# B&R Automation Studio project GAT (part 7)

#### Variables.var
```iecst
VAR
	MC_BR_ProcessConfig_AX : MC_BR_ProcessConfig; (*Function block to read and write the axis configuration*)
	MC_BR_ProcessConfig_ACP : MC_BR_ProcessConfig; (*Function block to read and write the ACOPOS configuration*)
	BaseAxConfig : ARRAY[0..1] OF McCfgAxType; (*Acopos configuration*)
	AcpAxConfig : ARRAY[0..1] OF McCfgAcpAxType; (*Acopos configuration*)
	uSelectedAxis : USINT; (*Selected Axis index*)
	sAxFeatures1 : ARRAY[0..2] OF STRING[255]; (*Axis features*)
	sAxFeatures2 : ARRAY[0..2] OF STRING[255]; (*Axis features*)
	uState : UINT; (*Read/Write state machine status*)
	bReadConfig : BOOL; (*Read config command*)
	bWriteConfig : BOOL; (*Write Acopos config command*)
	bSuccessRead : BOOL; (*Read config succeeded*)
	bErrorRead : BOOL; (*Read config failed*)
	bErrorWrite : BOOL; (*Write config failed*)
	bSuccessWrite : BOOL; (*Write config succeeded*)
	bSysReboot : BOOL;
	MpRecipeRegPar_M : ARRAY[0..3] OF MpRecipeRegPar;
	MC_BR_ProcessParam_ACP : MC_BR_ProcessParam;
END_VAR
```

#### Main.st
```iecst
//*********************************************************************************
//* Copyright: B&R Industrial Automation GmbH
//* This task let's the OEM change the ACOPOS configuration via the HMI
//*********************************************************************************

PROGRAM _INIT
	// FUB configuration: MC_BR_ProcessConfig for persistent configuration changes, MC_BR_ProcessParam for online configuration changes
    MC_BR_ProcessConfig_ACP.DataType := mcCFG_ACP_AX;

	AcpAxConfig[0].AxisFeatures.FeatureReference.DataAddress := ADR(AxFeatures1);
	AcpAxConfig[0].AxisFeatures.FeatureReference.NumberOfArrayElements := 3;
	AcpAxConfig[1].AxisFeatures.FeatureReference.DataAddress := ADR(AxFeatures2);
	AcpAxConfig[1].AxisFeatures.FeatureReference.NumberOfArrayElements := 3;

	MC_BR_ProcessConfig_AX.DataType := mcCFG_AX;

	MC_BR_ProcessParam_ACP.ExecutionMode := mcEM_IMMEDIATELY;
	MC_BR_ProcessParam_ACP.Mode := mcPPM_WRITE;

	// Register "Machine" category PVs
	MpRecipeRegPar_M[0].MpLink := ADR(gMpLinkRecipeXml);
	MpRecipeRegPar_M[0].Enable := TRUE;
	MpRecipeRegPar_M[0].Category := ADR('Machine');
	MpRecipeRegPar_M[0].PVName := ADR('ProcessCon:AcpAxConfig');
	MpRecipeRegPar_M[1].MpLink := ADR(gMpLinkRecipeXml);
	MpRecipeRegPar_M[1].Enable := TRUE;
	MpRecipeRegPar_M[1].Category := ADR('Machine');
	MpRecipeRegPar_M[1].PVName := ADR('ProcessCon:BaseAxConfig');
	MpRecipeRegPar_M[2].MpLink := ADR(gMpLinkRecipeXml);
	MpRecipeRegPar_M[2].Enable := TRUE;
	MpRecipeRegPar_M[2].Category := ADR('Machine');
	MpRecipeRegPar_M[2].PVName := ADR('ProcessCon:sAxFeatures1');
	MpRecipeRegPar_M[3].MpLink := ADR(gMpLinkRecipeXml);
	MpRecipeRegPar_M[3].Enable := TRUE;
	MpRecipeRegPar_M[3].Category := ADR('Machine');
	MpRecipeRegPar_M[3].PVName := ADR('ProcessCon:sAxFeatures2');

	// Activate RegPar FUBs
	WHILE NOT MpRecipeRegPar_M[0].Active DO
		MpRecipeRegPar_M[0]();
	END_WHILE
	WHILE NOT MpRecipeRegPar_M[1].Active DO
		MpRecipeRegPar_M[1]();
	END_WHILE
	WHILE NOT MpRecipeRegPar_M[2].Active DO
		MpRecipeRegPar_M[2]();
	END_WHILE
	WHILE NOT MpRecipeRegPar_M[3].Active DO
		MpRecipeRegPar_M[3]();
	END_WHILE

	// Trigger first read
	ReadConfig := TRUE;
	State := 0;
END_PROGRAM

PROGRAM _CYCLIC
	// Read/Write state machine
	CASE State OF
        0:
            // Idle
			IF MpRecipeRegPar_M[0].UpdateNotification THEN
				// Reset the address of sAxFeatures1/2
				AcpAxConfig[0].AxisFeatures.FeatureReference.DataAddress := ADR(AxFeatures1);
				AcpAxConfig[0].AxisFeatures.FeatureReference.NumberOfArrayElements := 3;
				AcpAxConfig[1].AxisFeatures.FeatureReference.DataAddress := ADR(AxFeatures2);
				AcpAxConfig[1].AxisFeatures.FeatureReference.NumberOfArrayElements := 3;

				// Write the configuration
				SelectedAxis := 0;
				WriteConfig := TRUE;
				ReadConfig := FALSE;
			ELSIF ReadConfig THEN
				// Set axis dependend configuration name
				IF SelectedAxis = 0 THEN
					brsstrcpy(ADR(MC_BR_ProcessConfig_ACP.Name), ADR('IF1.ST1/DriveConfiguration/Channel1'));
				ELSE
					brsstrcpy(ADR(MC_BR_ProcessConfig_ACP.Name), ADR('IF1.ST1/DriveConfiguration/Channel2'));
				END_IF
				AcpAxConfig[0].AxisFeatures.FeatureReference.DataAddress := ADR(AxFeatures1);
				AcpAxConfig[0].AxisFeatures.FeatureReference.NumberOfArrayElements := 3;
				AcpAxConfig[1].AxisFeatures.FeatureReference.DataAddress := ADR(AxFeatures2);
				AcpAxConfig[1].AxisFeatures.FeatureReference.NumberOfArrayElements := 3;

				MC_BR_ProcessConfig_ACP.DataAddress := ADR(AcpAxConfig[SelectedAxis]);
				MC_BR_ProcessConfig_AX.DataAddress := ADR(BaseAxConfig[SelectedAxis]);
				// Start loading
				MC_BR_ProcessConfig_ACP.Mode := mcPCM_LOAD;
				MC_BR_ProcessConfig_ACP.Execute := TRUE;
				ErrorRead := FALSE;
				SuccessRead := FALSE;
				State := 10;
			ELSIF WriteConfig THEN
				// Set axis dependend configuration name
				IF SelectedAxis = 0 THEN
					brsstrcpy(ADR(MC_BR_ProcessConfig_ACP.Name), ADR('IF1.ST1/DriveConfiguration/Channel1'));
					MC_BR_ProcessParam_ACP.Component := ADR(gAxisMaster);
				ELSE
					brsstrcpy(ADR(MC_BR_ProcessConfig_ACP.Name), ADR('IF1.ST1/DriveConfiguration/Channel2'));
					MC_BR_ProcessParam_ACP.Component := ADR(gAxisSlave);
				END_IF
				MC_BR_ProcessConfig_ACP.DataAddress := ADR(AcpAxConfig[SelectedAxis]);
				MC_BR_ProcessConfig_AX.DataAddress := ADR(BaseAxConfig[SelectedAxis]);
                MC_BR_ProcessParam_ACP.DataAddress := ADR(AcpAxConfig[SelectedAxis].MechanicalElements);
                // mcCFG_ACP_AX is not supported yet, therefore, transfer mech elements and homing parameters in two steps
				MC_BR_ProcessParam_ACP.DataType := mcCFG_ACP_MECH_ELM;
				// Copy direct homing position into the used homing mode, HMI is bound to direct homing position
				CASE AcpAxConfig[SelectedAxis].Homing.Mode.Type OF
					mcAHM_ABS:
						AcpAxConfig[SelectedAxis].Homing.Mode.Absolute.Position := AcpAxConfig[SelectedAxis].Homing.Mode.Direct.Position;
					mcAHM_ABS_CORR:
						AcpAxConfig[SelectedAxis].Homing.Mode.AbsoluteCorrection.Position := AcpAxConfig[SelectedAxis].Homing.Mode.Direct.Position;
					mcAHM_ABS_SW:
						AcpAxConfig[SelectedAxis].Homing.Mode.AbsoluteSwitch.Position := AcpAxConfig[SelectedAxis].Homing.Mode.Direct.Position;
					mcAHM_BLK_LAG_ERR:
						AcpAxConfig[SelectedAxis].Homing.Mode.BlockLagError.Position := AcpAxConfig[SelectedAxis].Homing.Mode.Direct.Position;
                    mcAHM_BLK_TORQ:
                        AcpAxConfig[SelectedAxis].Homing.Mode.BlockTorque.Position := AcpAxConfig[SelectedAxis].Homing.Mode.Direct.Position;
					mcAHM_DIST_C_MARKS:
						AcpAxConfig[SelectedAxis].Homing.Mode.DistanceCodedMarks.Position := AcpAxConfig[SelectedAxis].Homing.Mode.Direct.Position;
					mcAHM_DIST_C_MARKS_CORR:
						AcpAxConfig[SelectedAxis].Homing.Mode.DistanceCodedMarksCorrection.Position := AcpAxConfig[SelectedAxis].Homing.Mode.Direct.Position;
					mcAHM_LIM_SW:
						AcpAxConfig[SelectedAxis].Homing.Mode.LimitSwitch.Position := AcpAxConfig[SelectedAxis].Homing.Mode.Direct.Position;
					mcAHM_SW_GATE:
						AcpAxConfig[SelectedAxis].Homing.Mode.SwitchGate.Position := AcpAxConfig[SelectedAxis].Homing.Mode.Direct.Position;
				END_CASE;
				MC_BR_ProcessConfig_ACP.Mode := mcPCM_SAVE;
				MC_BR_ProcessConfig_ACP.Execute := TRUE;
				MC_BR_ProcessConfig_AX.Mode := mcPCM_SAVE;
				MC_BR_ProcessConfig_AX.Execute := TRUE;
				MC_BR_ProcessParam_ACP.Execute := TRUE;
				ErrorWrite := FALSE;
				SuccessWrite := FALSE;
				State := 20;
			END_IF

        10:
            // Read config
			IF MC_BR_ProcessConfig_ACP.Done OR MC_BR_ProcessConfig_ACP.Error THEN
				MC_BR_ProcessConfig_ACP.Execute := FALSE;
				// Copy homing position into the direct homing position, HMI is bound to direct homing position
				CASE AcpAxConfig[SelectedAxis].Homing.Mode.Type OF
					mcAHM_ABS:
						AcpAxConfig[SelectedAxis].Homing.Mode.Direct.Position := AcpAxConfig[SelectedAxis].Homing.Mode.Absolute.Position;
					mcAHM_ABS_CORR:
						AcpAxConfig[SelectedAxis].Homing.Mode.Direct.Position := AcpAxConfig[SelectedAxis].Homing.Mode.AbsoluteCorrection.Position;
					mcAHM_ABS_SW:
						AcpAxConfig[SelectedAxis].Homing.Mode.Direct.Position := AcpAxConfig[SelectedAxis].Homing.Mode.AbsoluteSwitch.Position;
					mcAHM_BLK_LAG_ERR:
						AcpAxConfig[SelectedAxis].Homing.Mode.Direct.Position := AcpAxConfig[SelectedAxis].Homing.Mode.BlockLagError.Position;
					mcAHM_BLK_TORQ:
						AcpAxConfig[SelectedAxis].Homing.Mode.Direct.Position := AcpAxConfig[SelectedAxis].Homing.Mode.BlockTorque.Position;
					mcAHM_DIST_C_MARKS:
						AcpAxConfig[SelectedAxis].Homing.Mode.Direct.Position := AcpAxConfig[SelectedAxis].Homing.Mode.DistanceCodedMarks.Position;
					mcAHM_DIST_C_MARKS_CORR:
						AcpAxConfig[SelectedAxis].Homing.Mode.Direct.Position := AcpAxConfig[SelectedAxis].Homing.Mode.DistanceCodedMarksCorrection.Position;
					mcAHM_LIM_SW:
						AcpAxConfig[SelectedAxis].Homing.Mode.Direct.Position := AcpAxConfig[SelectedAxis].Homing.Mode.LimitSwitch.Position;
					mcAHM_SW_GATE:
						AcpAxConfig[SelectedAxis].Homing.Mode.Direct.Position := AcpAxConfig[SelectedAxis].Homing.Mode.SwitchGate.Position;
				END_CASE;
				brsstrcpy(ADR(MC_BR_ProcessConfig_AX.Name), ADR(AcpAxConfig[SelectedAxis].AxisReference.Name));
				MC_BR_ProcessConfig_AX.Mode := mcPCM_LOAD;
				MC_BR_ProcessConfig_AX.Execute := TRUE;
				ErrorRead := FALSE;
				SuccessRead := TRUE;
				State := 11;
			ELSIF MC_BR_ProcessConfig_ACP.Error THEN
				MC_BR_ProcessConfig_ACP.Execute := FALSE;
				ErrorRead := TRUE;
				SuccessRead := FALSE;
				ReadConfig := FALSE;
				State := 0;
			END_IF

        11:
            // Read axis config
			IF MC_BR_ProcessConfig_AX.Done OR MC_BR_ProcessConfig_AX.Error THEN
				MC_BR_ProcessConfig_AX.Execute := FALSE;
				ErrorRead := MC_BR_ProcessConfig_AX.Error;
				SuccessRead := NOT bErrorRead;
				IF SelectedAxis = 0 THEN
					SelectedAxis := 1;
				ELSE
					ReadConfig := FALSE;
				END_IF
				State := 0;
			END_IF

        20:
            // Write config
			IF (MC_BR_ProcessConfig_ACP.Done OR MC_BR_ProcessConfig_ACP.Error)
				AND (MC_BR_ProcessConfig_AX.Done OR MC_BR_ProcessConfig_AX.Error)
				AND (MC_BR_ProcessParam_ACP.Done OR MC_BR_ProcessParam_ACP.Error) THEN
				MC_BR_ProcessConfig_ACP.Execute := FALSE;
				MC_BR_ProcessConfig_AX.Execute := FALSE;
				MC_BR_ProcessParam_ACP.Execute := FALSE;
				ErrorWrite := MC_BR_ProcessConfig_ACP.Error OR MC_BR_ProcessConfig_AX.Error OR MC_BR_ProcessParam_ACP.Error;
				SuccessWrite := NOT ErrorWrite;
				State := 21;
			END_IF

        21:
            // Write Homing config
			MC_BR_ProcessParam_ACP.DataAddress := ADR(AcpAxConfig[SelectedAxis].Homing);// mcCFG_ACP_AX is not supported yet, therefore, transfer mech elements and homing parameters in two steps
			MC_BR_ProcessParam_ACP.DataType := mcCFG_ACP_HOME;
			MC_BR_ProcessParam_ACP.Execute := TRUE;
			IF MC_BR_ProcessParam_ACP.Done OR MC_BR_ProcessParam_ACP.Error THEN
				MC_BR_ProcessParam_ACP.Execute := FALSE;
				ErrorWrite := bErrorWrite OR MC_BR_ProcessParam_ACP.Error;
				SuccessWrite := NOT bErrorWrite;
				State := 0;
				// Update the second axis, or finish
				IF SelectedAxis = 0 THEN
					SelectedAxis := 1;
				ELSE
					WriteConfig := FALSE;
				END_IF
			END_IF
	END_CASE;

	// PLC reboot
	IF SysReboot THEN
		SYSreset(TRUE, 1);
	END_IF

	// Function block calls
	MC_BR_ProcessConfig_ACP();
	MC_BR_ProcessConfig_AX();
	MC_BR_ProcessParam_ACP();
	MpRecipeRegPar_M[0]();
	MpRecipeRegPar_M[1]();
	MpRecipeRegPar_M[2]();
	MpRecipeRegPar_M[3]();
END_PROGRAM

PROGRAM _EXIT
	// Release mplink
	MpRecipeRegPar_M[0].Enable := FALSE;
	MpRecipeRegPar_M[1].Enable := FALSE;
	MpRecipeRegPar_M[2].Enable := FALSE;
	MpRecipeRegPar_M[3].Enable := FALSE;
	MpRecipeRegPar_M[0]();
	MpRecipeRegPar_M[1]();
	MpRecipeRegPar_M[2]();
	MpRecipeRegPar_M[3]();
END_PROGRAM
```

### Program Logical/Infrastructure/SysServices/IoBrowser (IEC) - Task to read the IO module structure and display the IO channels

#### Variables.var
```iecst
(*Io process related variables*)
VAR
	GatIoForcingHandler_0 : GatIoForcingHandler; (*Function block for Io handling (browser & forcing)*)
	IoModules : ARRAY[0..gatMAX_IDX_IO_MODULES] OF GatIoModulesType;
	pIoChannelTemp : REFERENCE TO GatIoChannelType;
	pIoChannel : REFERENCE TO GatIoChannelType;
END_VAR
(*Helper variables for mappView*)
VAR
	sStationList : ARRAY[0..gatMAX_IDX_IO_MODULES] OF STRING[80];
	sModuleList : ARRAY[0..gatMAX_IDX_IO_MODULES] OF STRING[80];
	sIoChannelList : ARRAY[0..gatMAX_IDX_IO_CHANNELS] OF STRING[80];
	sIoPvList : ARRAY[0..gatMAX_IDX_IO_CHANNELS] OF STRING[80];
	sIoValueList : ARRAY[0..gatMAX_IDX_IO_CHANNELS] OF STRING[20];
	iIoValueList : ARRAY[0..gatMAX_IDX_IO_CHANNELS] OF DINT;
	uStationIdx : UINT;
	uModuleIdx : UINT;
	uChannelIdx : UINT;
	sSelectedStation : STRING[80];
	uSelectedStation : UINT;
	uLastSelectedStation : UINT;
	uSelectedModule : UINT;
	uLastSelectedModule : UINT;
	uSelectedChannel : UINT;
	uLastSelectedChannel : UINT;
	sTableConfigChannels : STRING[200];
	sTableConfigStations : STRING[200];
	sTableConfig : STRING[200];
	sTempStationPath : STRING[80];
	bLastModuleInvisible : BOOL;
END_VAR
```

#### Main.st
```iecst
//*********************************************************************************
//* Copyright: B&R Industrial Automation GmbH
//* This program provides an Io browser and the related interface for
//* mappView widgets.
//*********************************************************************************

PROGRAM _INIT
	// Init Io handler
	GatIoForcingHandler_0.Enable := TRUE;
	GatIoForcingHandler_0.SelectedRefreshMode := TRUE;
	GatIoForcingHandler_0.IoModules := ADR(IoModules);

	// Init refresh selection
	FOR ChannelIdx := 0 TO gatMAX_IDX_IO_CHANNELS DO
		IoModules[0].IoChannels[ChannelIdx].IoForcing.RefreshActualValue := TRUE;
	END_FOR

	// Init Table configs for mappView
	brsstrcpy(ADR(TableConfig), ADR('{ "specRows": [{"from":0,"to":19, "visible":false}]}'));
	brsstrcpy(ADR(TableConfigStations), ADR('{ "specRows": [{"from":0,"to":19, "visible":false}]}'));
	brsstrcpy(ADR(TableConfigChannels), ADR('{ "specRows": [{"from":0,"to":31, "visible":false}]}'));

	// Init pointers
	IoChannel ACCESS ADR(IoModules[0].IoChannels[0]);
	IoChannelTemp ACCESS ADR(IoModules[0].IoChannels[0]);
END_PROGRAM

PROGRAM _CYCLIC
	// Action to prepare all necessary table configs etc for mappView according to the station/module selection
	mappViewAction;

	// Function block call
	GatIoForcingHandler_0();
END_PROGRAM

PROGRAM _EXIT
	// Disabled function block call
	GatIoForcingHandler_0.Enable := FALSE;
	GatIoForcingHandler_0();
END_PROGRAM
```

#### mappViewAction.st
```iecst
//*********************************************************************************
//* Copyright: B&R Industrial Automation GmbH
//* This action sets all the strings and pointers so that the mappView page can
//* present the IO information in a user friendly way
//********************************************************************************

ACTION mappViewAction:
	// Set pointers to the correct Forcing handler for easier interface to HMI
	IF (SelectedModule <> LastSelectedModule) OR (SelectedChannel <> LastSelectedChannel) THEN
		// Check range
		IF (SelectedModule <= gatMAX_IDX_IO_MODULES) AND (SelectedChannel <= gatMAX_IDX_IO_MODULES) THEN
			IF SelectedChannel >= IoModules[SelectedModule].NrOfIoChannels THEN
				SelectedChannel := 0;
			END_IF
			IoChannel ACCESS ADR(IoModules[SelectedModule].IoChannels[SelectedChannel]);
			IoChannelTemp ACCESS ADR(IoModules[SelectedModule].IoChannels[SelectedChannel]);
			brsmemset(ADR(IoChannelList), 0, SIZEOF(IoChannelList));
			brsmemset(ADR(IoPvList), 0, SIZEOF(IoPvList));
			brsmemset(ADR(IoValueList), 0, SIZEOF(IoValueList));
			brsmemset(ADR(TableConfigChannels), 0, SIZEOF(TableConfigChannels));
			FOR ChannelIdx := 0 TO gatMAX_IDX_IO_CHANNELS DO
				brsstrcpy(ADR(IoChannelList[ChannelIdx]), ADR(IoModules[SelectedModule].IoChannels[ChannelIdx].ChannelName));
				IF brsstrlen(ADR(IoChannelList[ChannelIdx])) = 0 THEN
					// Configure visible table entries
					brsstrcpy(ADR(TableConfigChannels), ADR('{ "specRows": [{"from":'));
					brsitoa(ChannelIdx, ADR(TableConfigChannels) + brsstrlen(ADR(TableConfigChannels)));
					brsstrcat(ADR(TableConfigChannels),  ADR(',"to":31, "visible":false}]}'));
					EXIT;
				END_IF
				brsstrcpy(ADR(IoPvList[ChannelIdx]), ADR('$$IAT/Audit/DP/'));
				IF brsstrlen(ADR(IoModules[SelectedModule].IoChannels[ChannelIdx].PvName)) = 0 THEN
					brsstrcat(ADR(IoPvList[ChannelIdx]), ADR('None'));
				ELSE
					brsstrcat(ADR(IoPvList[ChannelIdx]), ADR(IoModules[SelectedModule].IoChannels[ChannelIdx].PvName));
				END_IF
			END_FOR
			LastSelectedModule := SelectedModule;
			LastSelectedChannel := SelectedChannel;
		END_IF
		// Set Io refresh flags
		FOR ModuleIdx := 0 TO gatMAX_IDX_IO_MODULES DO
			FOR ChannelIdx := 0 TO gatMAX_IDX_IO_CHANNELS DO
				IoModules[ModuleIdx].IoChannels[ChannelIdx].IoForcing.RefreshActualValue := (ModuleIdx = SelectedModule);
			END_FOR
		END_FOR
	END_IF

	// Update IO values
	FOR ChannelIdx := 0 TO gatMAX_IDX_IO_CHANNELS DO
		IF IoModules[SelectedModule].IoChannels[ChannelIdx].IoForcing.ActualValue > 32767 THEN
			IoValueList[ChannelIdx] := IoModules[SelectedModule].IoChannels[ChannelIdx].IoForcing.ActualValue - 65536;
		ELSE
			IoValueList[ChannelIdx] := IoModules[SelectedModule].IoChannels[ChannelIdx].IoForcing.ActualValue;
		END_IF
		CASE IoModules[SelectedModule].IoChannels[ChannelIdx].Type OF
			IO_DIG_INPUT, IO_DIG_OUTPUT:
				IF (IoModules[SelectedModule].IoChannels[ChannelIdx].IoForcing.ActualValue = 1) THEN
					brsstrcpy(ADR(IoValueListString[ChannelIdx]), ADR('ON'));
				ELSE
					brsstrcpy(ADR(IoValueListString[ChannelIdx]), ADR('OFF'));
				END_IF
			IO_ANA_INPUT, IO_ANA_OUTPUT, IO_PWM_OUTPUT:
				brsftoa(DINT_TO_REAL(REAL_TO_DINT(DINT_TO_REAL(IoValueList[ChannelIdx]) / 32.767)) / 10, ADR(IoValueListString[ChannelIdx]));
				brsstrcat(ADR(IoValueListString[ChannelIdx]), ADR(' %'));
			IO_TEMP_INPUT:
				brsftoa(DINT_TO_REAL(IoValueList[ChannelIdx]) / 10, ADR(IoValueListString[ChannelIdx]));
				brsstrcat(ADR(IoValueListString[ChannelIdx]), ADR(' C'));
			ELSE
				brsitoa(IoValueList[ChannelIdx], ADR(IoValueListString[ChannelIdx]));
		END_CASE
	END_FOR

	// Init Io Module list when handler is ready
	IF EDGEPOS(GatIoForcingHandler_0.Ready) THEN
		brsmemset(ADR(TableConfigStations), 0, SIZEOF(TableConfig));
		brsmemset(ADR(StationList), 0, SIZEOF(StationList));
		// Init station list
		FOR ModuleIdx := 0 TO gatMAX_IDX_IO_MODULES DO
			IF FIND(RIGHT(IoModules[ModuleIdx].ModulePath, 6), '.') > 0 THEN
				brsmemset(ADR(TempStationPath), 0, SIZEOF(TempStationPath));
				brsstrcpy(ADR(TempStationPath), ADR('$$IAT/IoStations/'));
				brsmemcpy(ADR(TempStationPath) + brsstrlen(ADR(TempStationPath)), ADR(IoModules[ModuleIdx].ModulePath), brsstrlen(ADR(IoModules[ModuleIdx].ModulePath)) - 7 + FIND(RIGHT(IoModules[ModuleIdx].ModulePath, 6), '.'));
			END_IF
			FOR StationIdx := 0 TO gatMAX_IDX_IO_MODULES DO
				IF brsstrcmp(ADR(StationList[StationIdx]), ADR(TempStationPath)) = 0 THEN
					// Station already registered
					EXIT;
				END_IF
				IF brsstrlen(ADR(StationList[StationIdx])) = 0 THEN
					// Reached end of list, add new station
					brsstrcpy(ADR(StationList[StationIdx]), ADR(TempStationPath));
					EXIT;
				END_IF
			END_FOR
		END_FOR
		// Set station table configuration
		FOR StationIdx := 0 TO gatMAX_IDX_IO_MODULES DO
			IF brsstrlen(ADR(StationList[StationIdx])) = 0 THEN
				brsstrcpy(ADR(TableConfigStations), ADR('{ "specRows": [{"from":'));
				brsitoa(StationIdx, ADR(TableConfigStations) + brsstrlen(ADR(TableConfigStations)));
				brsstrcat(ADR(TableConfigStations),  ADR(',"to":'));
				brsstrcat(ADR(TableConfigStations),  ADR('19, "visible":false}]}'));
				EXIT;
			END_IF
		END_FOR
		// Trigger station selection
		SelectedStationIndex := 0;
		LastSelectedStationIndex := 1;
	END_IF

	// Init Module list after station selection
	IF SelectedStationIndex <> LastSelectedStationIndex THEN
		brsmemset(ADR(TableConfig), 0, SIZEOF(TableConfig));
		brsmemset(ADR(ModuleList), 0, SIZEOF(ModuleList));
		brsmemset(ADR(SelectedStation), 0, SIZEOF(SelectedStation));
		brsstrcpy(ADR(SelectedStation), ADR(StationList[SelectedStationIndex]) + brsstrlen(ADR('$$IAT/IoStations/')));
		// Init module list
		brsmemset(ADR(TableConfig), 0, SIZEOF(TableConfig));
		LastModuleInvisible := FALSE;
		FOR ModuleIdx := 0 TO gatMAX_IDX_IO_MODULES DO
			brsstrcpy(ADR(ModuleList[ModuleIdx]), ADR(IoModules[ModuleIdx].ModuleName));
			IF (FIND(IoModules[ModuleIdx].ModulePath, SelectedStation) = 0) THEN
				// Wrong station, make station invisible
				IF NOT LastModuleInvisible THEN
					IF brsstrlen(ADR(TableConfig)) = 0 THEN
						brsstrcpy(ADR(TableConfig), ADR('{ "specRows": [{"from":'));
					ELSE
						brsstrcat(ADR(TableConfig), ADR(', {"from":'));
					END_IF
					brsitoa(ModuleIdx, ADR(TableConfig) + brsstrlen(ADR(TableConfig)));
					brsstrcat(ADR(TableConfig),  ADR(',"to":'));
				END_IF
				LastModuleInvisible := TRUE;
			ELSE
				// Correct station, make module visible and select it if it's the first module of the station
				IF SelectedModule = LastSelectedModule THEN
					SelectedModule := ModuleIdx;
					LastSelectedModule := SelectedModule + 1;
				END_IF
				IF LastModuleInvisible THEN
					brsitoa(ModuleIdx - 1, ADR(TableConfig) + brsstrlen(ADR(TableConfig)));
					brsstrcat(ADR(TableConfig),  ADR(', "visible":false}'));
				END_IF
				LastModuleInvisible := FALSE;
			END_IF
			IF brsstrlen(ADR(ModuleList[ModuleIdx])) = 0 THEN
				// Reached end of modules, make rest of list invisible
				IF NOT LastModuleInvisible THEN
					IF brsstrlen(ADR(TableConfig)) = 0 THEN
						brsstrcpy(ADR(TableConfig), ADR('{ "specRows": [{"from":'));
					ELSE
						brsstrcat(ADR(TableConfig), ADR(', {"from":'));
					END_IF
					brsitoa(ModuleIdx, ADR(TableConfig) + brsstrlen(ADR(TableConfig)));
					brsstrcat(ADR(TableConfig),  ADR(',"to":'));
				END_IF
				brsstrcat(ADR(TableConfig),  ADR('19, "visible":false}]}'));
				EXIT;
			ELSIF ModuleIdx = gatMAX_IDX_IO_MODULES THEN
				// Reached end of modules, close table config
				IF LastModuleInvisible THEN
					brsitoa(ModuleIdx, ADR(TableConfig) + brsstrlen(ADR(TableConfig)));
					brsstrcat(ADR(TableConfig), ADR(', "visible":false}]}'));
				ELSE
					brsstrcat(ADR(TableConfig), ADR(']}'));
				END_IF
			END_IF
		END_FOR
	END_IF
	LastSelectedStationIndex := SelectedStationIndex;
END_ACTION
```

### TestCase.h
```c
/*
* Author: 		B+R
* Contents of this file are modified and extended
*/

/*
 * COPYRIGHT AND PERMISSION NOTICE
 *
 * Copyright (c) 2003 Embedded Unit Project
 *
 * All rights reserved.
 *
 * Permission is hereby granted, free of charge, to any person obtaining
 * a copy of this software and associated documentation files (the
 * "Software"), to deal in the Software without restriction, including
 * without limitation the rights to use, copy, modify, merge, publish,
 * distribute, and/or sell copies of the Software, and to permit persons
 * to whom the Software is furnished to do so, provided that the above
 * copyright notice(s) and this permission notice appear in all copies
 * of the Software and that both the above copyright notice(s) and this
 * permission notice appear in supporting documentation.
 *
 * THE SOFTWARE IS PROVIDED "AS IS", WITHOUT WARRANTY OF ANY KIND,
 * EXPRESS OR IMPLIED, INCLUDING BUT NOT LIMITED TO THE WARRANTIES OF
 * MERCHANTABILITY, FITNESS FOR A PARTICULAR PURPOSE AND NONINFRINGEMENT
 * OF THIRD PARTY RIGHTS. IN NO EVENT SHALL THE COPYRIGHT HOLDER OR
 * HOLDERS INCLUDED IN THIS NOTICE BE LIABLE FOR ANY CLAIM, OR ANY
 * SPECIAL INDIRECT OR CONSEQUENTIAL DAMAGES, OR ANY DAMAGES WHATSOEVER
 * RESULTING FROM LOSS OF USE, DATA OR PROFITS, WHETHER IN AN ACTION OF
 * CONTRACT, NEGLIGENCE OR OTHER TORTIOUS ACTION, ARISING OUT OF OR IN
 * CONNECTION WITH THE USE OR PERFORMANCE OF THIS SOFTWARE.
 *
 * Except as contained in this notice, the name of a copyright holder
 * shall not be used in advertising or otherwise to promote the sale,
 * use or other dealings in this Software without prior written
 * authorization of the copyright holder.
 *
 * $Id: TestCase.h,v 1.7 2004/02/10 16:19:29 arms22 Exp $
 */
#ifndef	__TESTCASE_H__
#define	__TESTCASE_H__

typedef struct __TestCase	TestCase;
typedef struct __TestCase	*TestCaseRef;/*compatible embUnit1.0*/

struct __TestCase
{
	TestImplement 	*isa;
	const char 		*name;
	unsigned long	mode;
	testStateEnum 	state;
	char 			abort;
	testStatusEnum (*setUp)(void);
	testStatusEnum (*tearDown)(void);
	testStatusEnum (*runTest)(void);

};

extern const TestImplement TestCaseImplement;

#define new_TestCase(name,setUp,tearDown,runTest)\
	{\
		(TestImplement*)&TestCaseImplement,\
		name,\
		0, \
		stateStart,\
		0,\
		setUp,\
		tearDown,\
		runTest\
	}

#endif/*__TESTCASE_H__*/
```

### UtMgr.var
```iecst
(********************************************************************
 * COPYRIGHT -- Bernecker + Rainer
 ********************************************************************
 * Library: UtMgr
 * File: UtMgr.var
 * Author: B+R
 ********************************************************************
 * Constants of library UtMgr
 ********************************************************************)
VAR CONSTANT
	utERR_GENERAL : DINT := -1057750784; (*General error, see help*)
	utMgrERR_INVALID_PARAM : DINT := -1057750783; (*Check parameters*)
	utMgrERR_TOO_MANY_TESTS : DINT := -1057750782; (*Too many UtMgrTestSuites enabled, disable unused instances*)
END_VAR
```

- Library Logical/Infrastructure/TS_UnitTest/Samples/Framework_Extension_With_Custom_Asserts/LibAssert1 (ANSIC) (no source held here)

### Program Logical/Infrastructure/TS_UnitTest/Samples/Framework_Extension_With_Custom_Asserts/SPL_AssertsEx

#### testSet_AssertsExt.c
```c
/********************************************************************
* COPYRIGHT -- Bernecker + Rainer
********************************************************************
* Program: SPL_AssertsEx
* Author: B+R
********************************************************************
* This test set shows the use of self created asserts.
* Asserts are implemented in the library LibAssert1.
********************************************************************/

#include <bur/plctypes.h>

#ifdef _DEFAULT_INCLUDES
#include <AsDefault.h>
#endif

#include "UnitTest.h"
#include "LibAssert1.h"

_TEST test_splAssert_ArrayOfRealValues(void)
{
	/* manual generated differences for demonstration of the SPL_ASSERT */
	FloatArray1[0] = 2;
	FloatArray2[0] = 2;

	FloatArray1[1] = 3;
	FloatArray2[1] = 1;

	FloatArray1[30] = 3.33;
	FloatArray2[30] = 1.11;

	FloatArrayDeltaForComparison[31] = 1; /* Within -> pass, equal -> failed */
	FloatArray1[31] = 3.33;
	FloatArray2[31] = 3.31;

	SPL_ASSERT_ARRAY_EQUAL_REAL(FloatArray1, FloatArray2, sizeof(FloatArray1) / sizeof(FloatArray1[0]) );
	SPL_ASSERT_ARRAY_REAL_WITHIN(FloatArrayDeltaForComparison, FloatArray1, FloatArray2, sizeof(FloatArray1) / sizeof(FloatArray1[0]) );
	TEST_DONE;
}

_TEST test_splAssert_Boundary()
{
	/* should fail */
	SPL_ASSERT_UPPER_BOUNDARY(2,4);

	/* should pass */
	SPL_ASSERT_UPPER_BOUNDARY(4,2);

	TEST_DONE;
}

/*
B+R UnitTest: This is generated code.
Do not edit! Do not move!
Description: UnitTest Testprogramm infrastructure (TestSet).
LastUpdated: 2015-04-14 12:04:07Z
By B+R UnitTest Helper Version: 2.0.0.0
*/
UNITTEST_FIXTURES(fixtures)
{
	new_TestFixture("test_splAssert_ArrayOfRealValues", test_splAssert_ArrayOfRealValues),
	new_TestFixture("test_splAssert_Boundary", test_splAssert_Boundary),
};

UNITTEST_CALLER_COMPLETE_EXPLICIT(testSet_AssertsExt, "testSet_AssertsExt", 0, 0, fixtures, 0, 0, 0);
```

### Program Logical/Infrastructure/TS_UnitTest/Samples/Framework_Features/SPL_Asserts (ANSIC)

#### README.txt
```
Please note

The samples in this program provides no good programming style!
They are solely for demonstrating the behavior of the framework.
Bad style:
	o	There is no test of any function or FB, just asserts failing or passing (depending on PV values)
	o	Expectations are variables and no constants
	o	Mulitple asserts per Test Case
```

#### testSuite.var
```iecst
(********************************************************************
 * COPYRIGHT -- Bernecker + Rainer
 ********************************************************************
 * Program: SPL_Asserts
 * Author: B+R
 ********************************************************************
 * Local variables of program SPL_Asserts
 * General variables
 ********************************************************************)
VAR
	Testsuite : UtMgrTestSuite := (Name:='SPL_Asserts',Description:='Shows asserts and usage',Type:=utMgrTEST_TYPE_C);
END_VAR
```

### Program Logical/Infrastructure/TS_UnitTest/Samples/Framework_Features/SPL_Behavior (ANSIC)

#### controlFlowVariables.var - Variables used in sub package "ControlFlow"
```iecst
(********************************************************************
 * COPYRIGHT -- Bernecker + Rainer
 ********************************************************************
 * Program: SPL_Behavior
 * File: controlFlowVariables.var
 * Author: B+R
 ********************************************************************
 * Local variables of program SPL_Behavior
 ********************************************************************)
VAR
	CounterInSet : DINT := 0;
	CounterInSet_LastChecked : DINT := 0;
	OutputString : STRING[200];
	CounterToStringBuffer : STRING[20] := '';
END_VAR
(*Warning "Warning : 'CountTestCaseRuns' defined but not used" can be ignored.
Warnings for this variable occurs when no LOG_FOR_EXEMPLIFICATION_TEST_BUSY is used inside a set. *)
VAR CONSTANT
	DEF_BUSY_STEPS : USINT := 2;
END_VAR
VAR
	CountTestCaseRuns : USINT := 0;
END_VAR
```

#### Package Logical/Infrastructure/TS_UnitTest/Samples/Framework_Features/SPL_Behavior/ControlFlow - Shows sequence of calls within test set (depending on the defined optional handles)

#### test_SetTestCases.c
```c
/********************************************************************
* COPYRIGHT -- Bernecker + Rainer
********************************************************************
* Program: SPL_Behavior
* Author: B+R
********************************************************************
* This test set shows the sequence of calls within a test set
* Add some busy conditions or test cases to see the changes.
********************************************************************/

#include <bur/plctypes.h>

#ifdef _DEFAULT_INCLUDES
#include <AsDefault.h>
#endif

#include "UnitTest.h"

#include "iHelperFunction.h"

void resetDataForTestSet_TestCases()
{
	resetDataForTestSet();
}

_CYCLIC_SET(void)
{
	LOG_FOR_EXEMPLIFICATION_CYCLIC_SET;

	return;
}

_TEST test_1(void)
{
	LOG_FOR_EXEMPLIFICATION_TEST_CASE_1;

	TEST_DONE;
}

_TEST test_2(void)
{
	LOG_FOR_EXEMPLIFICATION_TEST_CASE_2;

	TEST_DONE;
}

_TEST test_3(void)
{
	LOG_FOR_EXEMPLIFICATION_TEST_CASE_3;

	TEST_DONE;
}

/*
B+R UnitTest: This is generated code.
Do not edit! Do not move!
Description: UnitTest Testprogramm infrastructure (TestSet).
LastUpdated: 2015-04-14 12:03:48Z
By B+R UnitTest Helper Version: 2.0.0.0
*/
UNITTEST_FIXTURES(fixtures)
{
	new_TestFixture("test_1", test_1),
	new_TestFixture("test_2", test_2),
	new_TestFixture("test_3", test_3),
};

UNITTEST_CALLER_COMPLETE_EXPLICIT(test_SetTestCases, "test_SetTestCases", 0, 0, fixtures, 0, 0, cyclicSetCaller);
```

#### test_SetTestCases_SetSetup_SetTeardown.c
```c
/********************************************************************
* COPYRIGHT -- Bernecker + Rainer
********************************************************************
* Program: SPL_Behavior
* Author: B+R
********************************************************************
* This test set shows the sequence of calls within a test set
* Add some busy conditions or test cases to see the changes.
********************************************************************/

#include <bur/plctypes.h>

#ifdef _DEFAULT_INCLUDES
#include <AsDefault.h>
#endif

#include "UnitTest.h"

#include "iHelperFunction.h"

void resetDataForTestSet_SetSetupTeardown()
{
	resetDataForTestSet();
}

_CYCLIC_SET(void)
{
	LOG_FOR_EXEMPLIFICATION_CYCLIC_SET;
	return;
}

_SETUP_SET(void)
{
	LOG_FOR_EXEMPLIFICATION_SETUP_SET;
	TEST_DONE;
}

_TEARDOWN_SET(void)
{
	LOG_FOR_EXEMPLIFICATION_TEARDOWN_SET;
	TEST_DONE;
}

_TEST test_1(void)
{
	LOG_FOR_EXEMPLIFICATION_TEST_CASE_1;
	TEST_DONE;
}

_TEST test_2(void)
{
	LOG_FOR_EXEMPLIFICATION_TEST_CASE_2;
	TEST_DONE;
}

_TEST test_3(void)
{
	LOG_FOR_EXEMPLIFICATION_TEST_CASE_3;
	TEST_DONE;
}

/*
B+R UnitTest: This is generated code.
Do not edit! Do not move!
Description: UnitTest Testprogramm infrastructure (TestSet).
LastUpdated: 2015-04-14 12:03:48Z
By B+R UnitTest Helper Version: 2.0.0.0
*/
UNITTEST_FIXTURES(fixtures)
{
	new_TestFixture("test_1", test_1),
	new_TestFixture("test_2", test_2),
	new_TestFixture("test_3", test_3),
};

UNITTEST_CALLER_COMPLETE_EXPLICIT(test_SetTestCases_SetSetup_SetTeardown, "test_SetTestCases_SetSetup_SetTeardown", 0, 0, fixtures, setupSet, teardownSet, cyclicSetCaller);
```

### Library Logical/Infrastructure/TS_UnitTest/Samples/Tests_Program/SPLMyCalc (IEC) - Simple Calculator

#### SPLMyCalc.var
```iecst
(********************************************************************
 * COPYRIGHT --  Bernecker + Rainer
 ********************************************************************
 * Library: SPLMyCalc
 * File: SPLMyCalc.var
 * Author: B+R
 ********************************************************************
 * Constants of library SPLMyCalc
 ********************************************************************)
VAR CONSTANT
	splMyCalcERR_OUT_OF_RANGE : UINT := 50002;
	splMyCalcERR_NO_VALID_PARAM : UINT := 50001;
END_VAR
```

#### SPLMyCalc.st
```iecst
(********************************************************************
 * COPYRIGHT -- Bernecker + Rainer
 ********************************************************************
 * Library: SPLMyCalc
 * File: SPLMyCalc.st
 * Author: B+R
 ********************************************************************
 * Implementation of library SPLMyCalc
 ********************************************************************)

(* This can be used as a sample for  Test Driven Development (TDD)/ Test First Development
Steps (in a nutshell):
    o Define your API (FB, functions, ...)
		 this is already done for the FB MyCalc
	o Create a new test program (by using the template)
	o Write a test case (e.g. Addition) for this FB.
		The tests should describe the expected behavior.
	o Transfer the test program to the target and run the test in the test view
		The test case will fail
	o Implement this FB (Addition), build and transfer, then run the test again
		The test case will pass
	o Write next test (e.g. Subtraction).
	..
	o Write test for MIN / MAX (underflow/overflow)
   	o Run the tests to verify your implementation.

Note:
	The sample test program in SPL_MyCalcLib_C provides some test cases using this FB.

 *)
FUNCTION_BLOCK MyCalculator

	Status := ERR_NOTIMPLEMENTED;

END_FUNCTION_BLOCK
```

### Package Logical/Infrastructure/TS_UnitTest/Samples/Tests_Program/Tests_MyCalcLib_C - Tests SPLMyCalc with library "UnitTest"

### Program Logical/Infrastructure/TS_UnitTest/Samples/Tests_Program/Tests_MyCalcLib_C/SPL_CalcTest

#### autoGeneratedFile.c
```c
/*
B+R UnitTest: This is generated code.
Do not edit! Do not move!
Description: UnitTest Testprogramm infrastructure (List of TestSets).
LastUpdated: 2015-04-14 12:04:18Z
By B+R UnitTest Helper Version: 2.0.0.0
*/
#include "UnitTest.h"

UNITTEST_TESTSET_DECLARATION  testSet_MyCalcLib_Addition;
UNITTEST_TESTSET_DECLARATION  testSet_MyCalcLib_Subtraction;
UNITTEST_TESTSET_DECLARATION  testSet_MyCalcLib_Mult_Div;

UNITTEST_TESTSET_FIXTURES(utTestSets)
{
	new_TestSet(testSet_MyCalcLib_Addition),
	new_TestSet(testSet_MyCalcLib_Subtraction),
	new_TestSet(testSet_MyCalcLib_Mult_Div),
};
UNTITTEST_TESTSET_HANDLER();
```

### Program Logical/Infrastructure/TS_UnitTest/Samples/Tests_Program/Tests_MyCalcLib_C/SPL_CalcTest_Variants

#### testSet_MyCalcLib_Subtraction.c
```c
/********************************************************************
 * COPYRIGHT -- Bernecker + Rainer
 ********************************************************************
 * Program: SPL_CalcTest_Variants
 * Author: B+R
 ********************************************************************
 * Test set implementation
 ********************************************************************/

#include <bur/plctypes.h>

#ifdef _DEFAULT_INCLUDES
#include <AsDefault.h>
#endif

#include "UnitTest.h"

_TEST test_Subtract(void)
{
	/* initialize functionblock parameters */
	instMyCalc.CalcOperator = splMyCalcOPERATOR_SUBTRACT;
	instMyCalc.Param1   = 4;
	instMyCalc.Param2   = 2;
	/* call synchron functionblock */
	MyCalculator(&instMyCalc);

	/* check result */
	TEST_ASSERT_EQUAL_INT(2, instMyCalc.Result);
	TEST_ASSERT_EQUAL_INT(ERR_OK, instMyCalc.Status);

	/* test is done */
	TEST_DONE;
}

_TEST test_Subtract_negResult(void)
{
	/* initialize functionblock parameters */
	instMyCalc.CalcOperator = splMyCalcOPERATOR_SUBTRACT;
	instMyCalc.Param1   = 6;
	instMyCalc.Param2   = 8;
	/* call synchron functionblock */
	MyCalculator(&instMyCalc);

	/* check result */
	TEST_ASSERT_EQUAL_INT(-2, instMyCalc.Result);
	TEST_ASSERT_EQUAL_INT(ERR_OK, instMyCalc.Status);

	/* test is done */
	TEST_DONE;
}

_TEST test_Subtract_zeroResult(void)
{
	/* initialize functionblock parameters */
	instMyCalc.CalcOperator = splMyCalcOPERATOR_SUBTRACT;
	instMyCalc.Param1   = 6;
	instMyCalc.Param2   = 6;
	/* call synchron functionblock */
	MyCalculator(&instMyCalc);

	/* check result */
	TEST_ASSERT_EQUAL_INT(0, instMyCalc.Result);
	TEST_ASSERT_EQUAL_INT(ERR_OK, instMyCalc.Status);

	/* test is done */
	TEST_DONE;
}

_TEST test_Subtract_boundaryArea_expect_MIN(void)
{
	/* initialize functionblock parameters */
	instMyCalc.CalcOperator = splMyCalcOPERATOR_SUBTRACT;
	instMyCalc.Param1   = -1;
	instMyCalc.Param2   = 32768;
	/* call synchron functionblock */
	MyCalculator(&instMyCalc);

	/* check result */
	TEST_ASSERT_EQUAL_INT(-32768, instMyCalc.Result);
	TEST_ASSERT_EQUAL_INT(splMyCalcERR_OUT_OF_RANGE, instMyCalc.Status);

	/* test is done */
	TEST_DONE;
}

/*
B+R UnitTest: This is generated code.
Do not edit! Do not move!
Description: UnitTest Testprogramm infrastructure (TestSet).
LastUpdated: 2015-04-14 12:04:18Z
By B+R UnitTest Helper Version: 2.0.0.0
*/
UNITTEST_FIXTURES(fixtures)
{
	new_TestFixture("test_Subtract", test_Subtract),
	new_TestFixture("test_Subtract_negResult", test_Subtract_negResult),
	new_TestFixture("test_Subtract_zeroResult", test_Subtract_zeroResult),
	new_TestFixture("test_Subtract_boundaryArea_expect_MIN", test_Subtract_boundaryArea_expect_MIN),
};

UNITTEST_CALLER_COMPLETE_EXPLICIT(testSet_MyCalcLib_Subtraction, "testSet_MyCalcLib_Subtraction", 0, 0, fixtures, 0, 0, 0);
```

#### testSet_MyCalcLib_Subtraction_variantA.c
```c
/********************************************************************
 * COPYRIGHT -- Bernecker + Rainer
 ********************************************************************
 * Program: SPL_CalcTest_Variants
 * Author: B+R
 ********************************************************************
 * Test set implementation
 ********************************************************************/

#include <bur/plctypes.h>

#ifdef _DEFAULT_INCLUDES
#include <AsDefault.h>
#endif

#include "UnitTest.h"

/* To check multiple subtraction combinations without code duplication a helper function can be created.

Note: If an check (assert) is extracted into a helper function, the error report do not contain information about the parameters this helper function was called. For some use cases, this will be acceptable/OK for others not.
	See test_Subtract_MultipleCases()
One option to avoid this is to create multiple Test Cases each calling the same helper function once but with different parameters.
	See test_Subtract_1() and test_Subtract_boundaryArea_expect_MIN()  */
void verify_subtract(INT par1, INT par2 , DINT expectResult)
{
	instMyCalc.CalcOperator = splMyCalcOPERATOR_SUBTRACT;
	instMyCalc.Param1   = par1;
	instMyCalc.Param2   = par2;
	/* call synchron functionblock */
	MyCalculator(&instMyCalc);
	/* check result */
	TEST_ASSERT_EQUAL_INT(expectResult, instMyCalc.Result);
	TEST_ASSERT_EQUAL_INT(ERR_OK, instMyCalc.Status);
}

_TEST test_Subtract(void)
{
	verify_subtract(4, 2,2);

	/* test is done */
	TEST_DONE;
}

_TEST test_Subtract_negResult(void)
{
	verify_subtract(6, 8, -2);

	/* test is done */
	TEST_DONE;
}

_TEST test_Subtract_zeroResult(void)
{
	verify_subtract(6, 6, 0);

	/* test is done */
	TEST_DONE;
}

/* This test isn't reduced as there is (currently) no argument for  instMyCalc.Status  */
_TEST test_Subtract_boundaryArea_expect_MIN(void)
{
	/* initialize functionblock parameters */
	instMyCalc.CalcOperator = splMyCalcOPERATOR_SUBTRACT;
	instMyCalc.Param1   = -1;
	instMyCalc.Param2   = 32768;
	/* call synchron functionblock */
	MyCalculator(&instMyCalc);

	/* check result */
	TEST_ASSERT_EQUAL_INT(-32768, instMyCalc.Result);
	TEST_ASSERT_EQUAL_INT(splMyCalcERR_OUT_OF_RANGE, instMyCalc.Status);

	/* test is done */
	TEST_DONE;
}

/*
B+R UnitTest: This is generated code.
Do not edit! Do not move!
Description: UnitTest Testprogramm infrastructure (TestSet).
LastUpdated: 2015-04-14 12:04:18Z
By B+R UnitTest Helper Version: 2.0.0.0
*/
UNITTEST_FIXTURES(fixtures)
{
	new_TestFixture("test_Subtract", test_Subtract),
	new_TestFixture("test_Subtract_negResult", test_Subtract_negResult),
	new_TestFixture("test_Subtract_zeroResult", test_Subtract_zeroResult),
	new_TestFixture("test_Subtract_boundaryArea_expect_MIN", test_Subtract_boundaryArea_expect_MIN),
};

UNITTEST_CALLER_COMPLETE_EXPLICIT(testSet_MyCalcLib_Subtraction_variantA, "testSet_MyCalcLib_Subtraction_variantA", 0, 0, fixtures, 0, 0, 0);
```

### Steps.txt
```
Precondition: UnitTest Libraries are added to current active configuration
	(See AS help:  Solutions - Technology solutions - Unit test - Getting started - Adjusting the target configuration)

1. 	Copy template program
2. 	Rename the copy of the template program
3. 	Rename TestSuite.Name
4. 	Copy test set template

5. 	Implement test case
6. 	Copy batch file "Update_TestPrograms_in_current_location.bat" if it is not already in destination package
7. 	Double click batch file

8. 	Add test program to active software configuration
9.	Compile & transfer
10. Refresh test list in the test view
11. Run test
```

### Program Logical/Infrastructure/TS_UnitTest/Templates/HelperTool_Supported/utTemplate_automated (ANSIC)

#### testSuite.c
```c
/********************************************************************
 * COPYRIGHT --
 ********************************************************************
 * Program: -
 * Author:
 * Created:
 ********************************************************************
 * Test registration and handshake
 ********************************************************************/

#include <bur/plctypes.h>

#ifdef _DEFAULT_INCLUDES
#include <AsDefault.h>
#endif

#include "UnitTest.h"

void _INIT initTestSuite(void)
{
	utInit(&Testsuite);
}

void _CYCLIC cyclicWithTest(void)
{
	utCyclic(&Testsuite);
}

void _EXIT exitTestSuite(void)
{
	utExit(&Testsuite);
}
```

#### autoGeneratedFile.c - Auto generated code - list of all test sets in the program
```c
/* This content will be auto updated by the helper tool */

#include "UnitTest.h"

UNITTEST_TESTSET_FIXTURES (utTestSets)
{
	{
		0
	}
};
UNTITTEST_TESTSET_HANDLER();
```

- Program Logical/Infrastructure/TS_UnitTest/Templates/NoToolSupport/utTemplate_manual (ANSIC) (no source held here)

### Program Logical/Infrastructure/Alarm/AlarmMgt

#### Alarm.typ
```iecst
TYPE
	MachineDigitalInputs_type : 	STRUCT  (*Safety related digital inputs of the machine*)
		EmergencyStop : ARRAY[0..MAX_IDX_ESTOP]OF BOOL; (*Emergency stop signal*)
		SafetyDoor : ARRAY[0..MAX_IDX_SAFETY_DOOR]OF BOOL; (*Safety door signal*)
		AcknowledgeAlarms : BOOL;
	END_STRUCT;
	AlarmExamples_typ : 	STRUCT
		LevelMonitoring : INT := 50;
		DeviationMonitoring : INT := 15;
		DeviationMonitoringSetpoint : INT := 15;
		RateOfChange : INT;
		SnippetValue : INT := 10;
		ControlExample : BOOL;
	END_STRUCT;
	ActiveAlarmState_enum :
		(
		ACTIVE_ALARM_WAIT,
		ACTIVE_ALARM_QUERY,
		ACTIVE_ALARM_NEXT
		);
	AlarmType : 	STRUCT
		Active : BOOL;
		Acknowledged : BOOL;
		Scope : WSTRING[80];
		Name : STRING[80];
		Message : WSTRING[255];
		AdditionalInfo : WSTRING[255];
		TimeStamp : DATE_AND_TIME;
		Code : UDINT;
		Severity : UDINT;
	END_STRUCT;
	AlarmQueryType : 	STRUCT
		Next : BOOL;
		State : ActiveAlarmState_enum;
		LastActiveAlarmUpdateCount : UDINT;
		ActiveAlarmUpdateCount : UDINT;
		Alarms : ARRAY[0..19]OF AlarmType;
	END_STRUCT;
	AlarmHmiInterface_type : 	STRUCT
		Commands : AlarmCommands_type;
		Status : AlarmStatus_type;
	END_STRUCT;
	AlarmStatus_type : 	STRUCT
		AlarmHistSortCfg : STRING[1000];
		AlarmHistFilterCfg : STRING[1000];
		AlarmSortCfg : STRING[1000];
		AlarmFilterCfg : STRING[1000];
	END_STRUCT;
	AlarmCommands_type : 	STRUCT
		ExportAlarms : BOOL;
	END_STRUCT;
END_TYPE
```

#### Alarm.var
```iecst
(********************************************************************
 * COPYRIGHT -- Bernecker + Rainer
 ********************************************************************
 * Program: FolderHandling
 * File: FolderHandling.var
 * Author: Bernecker + Rainer
 * Created: December , 2020
 ********************************************************************
 * Local variables of program AlarmManagement
 ********************************************************************)
(*Function Blocks--------------------------------------------------------------------------------------------------------------------*)
VAR
	hmiAlarmX : AlarmHmiInterface_type;
	MpAlarmXHistory_0 : MpAlarmXHistory; (*MpAlarmXHistory instance*)
	MpAlarmXHistoryUI_0 : MpAlarmXHistoryUI; (*MpAlarmXHistoryUI instance*)
	MpAlarmXListUI_0 : MpAlarmXListUI; (*MpAlarmXList instance*)
	MpAlarmXCore_0 : MpAlarmXCore; (*MpAlarmXCore instance*) (*ChangeStyleAlarmButton : USINT := 0; (*changeStyle of a AlarmFlyout in mappView*)
	DirCreate_New : DirCreate;
END_VAR
(*Alarm Management Variables------------------------------------------------------------------------------------------------*)
VAR
	Index : USINT; (*Index to loop through alarm list*)
	MaxIndex : USINT; (*Maximum index for the alarm list*)
	uInstanceID : UINT; (*Instance ID*)
	MpAlarmXListUIConnect : MpAlarmXListUIConnectType := (0); (*AlarmVideo : WSTRING[255] := "";
	AlarmInfo : BOOL := 0;*)
	MpAlarmXHistoryUIConnect : MpAlarmXHistoryUIConnectType; (*AlarmX History connection to UI*)
	AlarmQuery : {REDUND_UNREPLICABLE} AlarmQueryType; (*Query Results*)
	QueryActiveAlarms : {REDUND_UNREPLICABLE} MpAlarmXQuery; (*MpAlarmXQuery instance*)
END_VAR
(*Safety Inputs*)
VAR
	SafetyInputs : MachineDigitalInputs_type;
END_VAR
(*Defines*)
VAR CONSTANT
	MAX_IDX_ESTOP : UINT := 2;
	MAX_IDX_SAFETY_DOOR : UINT := 5;
	LOCAL_FOLDER : STRING[10] := 'AlarmX';
END_VAR
(*Examples*)
VAR
	CommissioningModeActive : {REDUND_UNREPLICABLE} BOOL; (*Inhibits the Alarms[0] alarm*)
	Alarms : {REDUND_UNREPLICABLE} ARRAY[0..99] OF BOOL; (*Array of active alarm*)
	AlarmExamples : {REDUND_UNREPLICABLE} AlarmExamples_typ; (*Sample alarms for different monitoring types*)
	MpAlarmXControlExampleFB : {REDUND_UNREPLICABLE} MpAlarmXAlarmControl; (*MpAlarmXAlarmControl instance*)
END_VAR
```

#### Alarm.st
```iecst
	(*********************************************************************************
	* Copyright: B&R Industrial Automation GmbH
	* Author:    B&R Industrial Automation GmbH
	* Created:   30. Sep 2020/08:00
	* Description: Tasks for alarm control. The Alarm Management handling is done in this task.
	*********************************************************************************)
PROGRAM _INIT

	(*Create folder for this component on the user file device*)
	DirCreate_New(enable := TRUE, pDevice := ADR('userPartition'), pName := ADR(LOCAL_FOLDER));

	(*Check if folder already exist and if so disabled the function block call*)
	IF DirCreate_New.status = fiERR_DIR_ALREADY_EXIST THEN
		DirCreate_New(enable := FALSE);
	END_IF

	(* Init function blocks *)
    MpAlarmXCore_0.Enable := TRUE;
    MpAlarmXCore_0.MpLink := ADR(gAlarmXMpLink);
    MpAlarmXCore_0();

    MpAlarmXHistory_0.Enable := TRUE;
    MpAlarmXHistory_0.DeviceName := ADR('mappAlarmX');
    MpAlarmXHistory_0.MpLink := ADR(gAlarmXHistoryMpLink);
    MpAlarmXHistory_0();

	MpAlarmXListUI_0.Enable := TRUE;
    MpAlarmXListUI_0.UISetup.AlarmListScrollWindow := 10;
    MpAlarmXListUI_0.UISetup.AlarmListSize := 50;
	MpAlarmXListUI_0.UISetup.TimeStampPattern := '%Y %m %d %H:%M:%S';

    MpAlarmXHistoryUI_0.Enable := TRUE;
    MpAlarmXHistoryUI_0.UISetup.AlarmListScrollWindow := 10;
    MpAlarmXHistoryUI_0.UISetup.AlarmListSize := (SIZEOF(MpAlarmXListUIConnect.AlarmList.InstanceID)/SIZEOF(MpAlarmXListUIConnect.AlarmList.InstanceID[0]));
    MpAlarmXHistoryUI_0.UISetup.TimeStampPattern := '%Y %m %d %H:%M:%S';

    AlarmSamples;

	AlarmFilterCfg;
	AlarmSortCfg;
	AlarmHistFilterCfg;
	AlarmHistSortCfg;

END_PROGRAM

PROGRAM _CYCLIC

	(* Acknowledge Button *)
    IF EDGEPOS(SafetyInputs.AcknowledgeAlarms) THEN
        MpAlarmXListUIConnect.AcknowledgeAll := TRUE;
	END_IF

	(* Call all actions *)
    GetBacktraceInformation;
    ExecuteQuery;
    AlarmHandling;
    AlarmSamples;

    (* Check if any reactions are active *)
    IF MpAlarmXCheckReaction(gAlarmXMpLink, 'Error') THEN
        (* Error is active *)
    ELSIF MpAlarmXCheckReaction(gAlarmXMpLink, 'Warning') THEN
        (* Warning is active *)
	ELSIF MpAlarmXCheckReaction(gAlarmXMpLink, 'Info') THEN
        (* Info is active *)
	END_IF

	IF (ExportAlarms = TRUE) THEN
		ExportAlarms := FALSE;
		MpAlarmXHistory_0.Export := TRUE;
	END_IF

    (* Function block calls *)
    MpAlarmXCore_0.MpLink := ADR(gAlarmXMpLink);
    MpAlarmXCore_0();
    MpAlarmXListUI_0.MpLink := ADR(gAlarmXMpLink);
    MpAlarmXListUI_0.UIConnect := ADR(MpAlarmXListUIConnect);
    MpAlarmXListUI_0();
    MpAlarmXHistory_0.MpLink := ADR(gAlarmXHistoryMpLink);
	MpAlarmXHistory_0();
	MpAlarmXHistoryUI_0.MpLink := ADR(gAlarmXHistoryMpLink);
    MpAlarmXHistoryUI_0.UIConnect := ADR(MpAlarmXHistoryUIConnect);
	MpAlarmXHistoryUI_0();

	IF ((MpAlarmXHistory_0.Export = TRUE) AND (MpAlarmXHistory_0.CommandDone = TRUE)) THEN
		MpAlarmXHistory_0.Export := FALSE;
	END_IF

    (* Error reset *)
    IF NOT MpAlarmXCore_0.Error THEN
        MpAlarmXCore_0.ErrorReset := FALSE;
    END_IF
    IF NOT MpAlarmXListUI_0.Error THEN
        MpAlarmXListUI_0.ErrorReset := FALSE;
    END_IF
    IF NOT MpAlarmXHistory_0.Error THEN
        MpAlarmXHistory_0.ErrorReset := FALSE;
    END_IF
    IF NOT MpAlarmXHistoryUI_0.Error THEN
        MpAlarmXHistoryUI_0.ErrorReset := FALSE;
    END_IF

END_PROGRAM

PROGRAM _EXIT
	(* Reset function blocks to unlink mapp links *)
    MpAlarmXCore_0.Enable := FALSE;
    MpAlarmXListUI_0.Enable := FALSE;
    MpAlarmXHistory_0.Enable := FALSE;
	MpAlarmXHistoryUI_0.Enable := FALSE;
	QueryActiveAlarms.Enable := FALSE;
    MpAlarmXCore_0();
    MpAlarmXListUI_0();
    MpAlarmXHistory_0();
    MpAlarmXHistoryUI_0();
    QueryActiveAlarms();

END_PROGRAM
```

#### AlarmHandling.st
```iecst
ACTION AlarmHandling:

    // CommissioningModeActive will inhibit Alarms[0], see mpAlarmX configuration (must enable Advanced Features)
    // CommissioningModeActive = TRUE will inhibit Alarms[0], = FALSE will NOT inhibit Alarms[0]
    CommissioningModeActive;

    Alarms[0];
//    Alarms[1] := ;
//    Alarms[2] := ;
//    Alarms[3] := ;
//    Alarms[4] := ;
//    Alarms[5] := ;
//    Alarms[6] := ;
//    Alarms[7] := ;
//    Alarms[8] := ;
//    Alarms[9] := ;
//
//    Alarms[10] := ;
//    Alarms[11] := ;
//    Alarms[12] := ;
//    Alarms[13] := ;
//    Alarms[14] := ;
//    Alarms[15] := ;
//    Alarms[16] := ;
//    Alarms[17] := ;
//    Alarms[18] := ;
//    Alarms[19] := ;

END_ACTION
```

#### AlarmSamples.st
```iecst
ACTION AlarmSamples:

    // Call all variables that are needed for the alarm examples and explain all examples in comments

    // If AlarmExamples.LevelMonitoring gets less than 20 or more than 80, the LevelMonitoringExample alarm will trigger
	// The Low limit is 20. The LowLow limit is 10. The High limit is 80. The HighHigh limit is 90.
	AlarmExamples.LevelMonitoring;
	// If AlarmExamples.DeviationMonitoring deviates from the setpoint (AlarmExamples.DeviationMonitoringSetpoint) by more than 5
	// units in either direction, the DeviationMonitoringExample alarm will trigger
    AlarmExamples.DeviationMonitoring;
	AlarmExamples.DeviationMonitoringSetpoint;
    // If AlarmExamples.RateOfChange increases at a rate of more than 5 units per second, the RateOfChangeExample alarm will trigger
	AlarmExamples.RateOfChange;
	//If AlarmExamples.SnippetValue gets between 50 and 100, an alarm will trigger and the current value will be shown in the alarm text
    AlarmExamples.SnippetValue;

    MpAlarmXControlExampleFB.MpLink := ADR(gAlarmXMpLink);
    MpAlarmXControlExampleFB.Enable := TRUE;
    MpAlarmXControlExampleFB.Name := ADR('MpAlarmXControlExample');
    MpAlarmXControlExampleFB.Set := AlarmExamples.ControlExample;
    MpAlarmXControlExampleFB();

END_ACTION
```

#### Backtrace.st
```iecst
ACTION GetBacktraceInformation:

    MaxIndex := (SIZEOF(MpAlarmXListUIConnect.AlarmList.InstanceID)/SIZEOF(MpAlarmXListUIConnect.AlarmList.InstanceID[0])) - 1;
    // Find selected alarm in order to show backtrace information
    FOR Index := 0 TO MaxIndex DO
        IF (MpAlarmXCore_0.PendingAlarms = 0) THEN
            // No pending alarms, reset instance id
            uInstanceID := 0;
            EXIT;
        END_IF

        IF (MpAlarmXListUIConnect.AlarmList.InstanceID[Index] = uInstanceID) THEN
            // Found alarm
            MpAlarmXListUIConnect.AlarmList.SelectedIndex := Index;
            EXIT;
        END_IF

        IF (MpAlarmXListUIConnect.AlarmList.InstanceID[Index] = 0) THEN
            IF (MpAlarmXCore_0.PendingAlarms > Index) THEN
                // Alarm not found, List can page up
                MpAlarmXListUIConnect.AlarmList.PageUp := TRUE;
            END_IF
			EXIT;
        ELSIF (Index = MaxIndex) THEN
            // Alarm not found, List can page down
            MpAlarmXListUIConnect.AlarmList.PageDown := TRUE;
        END_IF
	END_FOR

END_ACTION
```

#### ExecuteQuery.st
```iecst
ACTION ExecuteQuery:

    QueryActiveAlarms.MpLink := ADR(gAlarmXMpLink);
    QueryActiveAlarms.Enable := TRUE;
    QueryActiveAlarms.Name := ADR('ActiveAlarms');
    QueryActiveAlarms.Language := ADR('en');
    QueryActiveAlarms();

    CASE (AlarmQuery.State) OF
        ACTIVE_ALARM_WAIT:
            IF (AlarmQuery.LastActiveAlarmUpdateCount <> AlarmQuery.ActiveAlarmUpdateCount) THEN
                brsmemset(ADR(AlarmQuery.Alarms[0]), 0, SIZEOF(AlarmQuery.Alarms));
                AlarmQuery.LastActiveAlarmUpdateCount := AlarmQuery.ActiveAlarmUpdateCount;
                QueryActiveAlarms.Execute := TRUE;
                AlarmQuery.State := ACTIVE_ALARM_QUERY;
            END_IF

        ACTIVE_ALARM_QUERY:
            IF ((QueryActiveAlarms.CommandDone = TRUE) AND (QueryActiveAlarms.Info.HasMoreRows = FALSE)) THEN
                QueryActiveAlarms.Execute := FALSE;
                QueryActiveAlarms.Next := FALSE;
                AlarmQuery.State := ACTIVE_ALARM_WAIT;
            ELSIF ((QueryActiveAlarms.CommandDone = TRUE) AND (QueryActiveAlarms.Info.HasMoreRows = TRUE)) THEN
                QueryActiveAlarms.Next := FALSE;
                AlarmQuery.State := ACTIVE_ALARM_NEXT;
            END_IF

        ACTIVE_ALARM_NEXT:
            IF (AlarmQuery.Next = TRUE) THEN
                brsmemset(ADR(AlarmQuery.Alarms[0]), 0, SIZEOF(AlarmQuery.Alarms));
                AlarmQuery.Next := FALSE;
                QueryActiveAlarms.Next := TRUE;
                AlarmQuery.State := ACTIVE_ALARM_QUERY;
            END_IF

    END_CASE

END_ACTION
```

- Program Logical/Infrastructure/AxisTemplate/AxisMgr (IEC) - Axis control (no source held here)

### Package Logical/Infrastructure/AxisTemplate/UnitTests - Multiple variants of valid test sets

### Program Logical/Infrastructure/AxisTemplate/UnitTests/prototypeTest (ANSIC)

#### variables.var - Name the suite and add PVs for the program
```iecst
(********************************************************************
 * COPYRIGHT --
 ********************************************************************
 * Program: utTemplate_automated
 * File: variables.var
 * Author: -
 * Created: -
 ********************************************************************
 * Local variables of program utTemplate_automated
 ********************************************************************)
(*Describe the test*)
VAR
	Testsuite : {REDUND_UNREPLICABLE} UtMgrTestSuite := (Enable:=TRUE,Name:='prototype',Description:='automated tests for prototype axis',Type:=utMgrTEST_TYPE_C);
	lastTestCase : {REDUND_UNREPLICABLE} STRING[80];
	lastTestSet : {REDUND_UNREPLICABLE} STRING[80];
END_VAR
(*Variables used in the tests*)
VAR
	AxisControl : {REDUND_UNREPLICABLE} AxisControlType;
	absVelocity : {REDUND_UNREPLICABLE} REAL;
	testState : {REDUND_UNREPLICABLE} testState_enum;
END_VAR
```

#### testSuite.c
```c
/********************************************************************
 * COPYRIGHT --
 ********************************************************************
 * Program: -
 * Author:
 * Created:
 ********************************************************************
 * Test registration and handshake
 ********************************************************************/

#include <bur/plctypes.h>

#ifdef _DEFAULT_INCLUDES
#include <AsDefault.h>
#endif

#include "UnitTest.h"

void _INIT initTestSuite(void)
{
	utInit(&Testsuite);
}

void _CYCLIC cyclicWithTest(void)
{
	utCyclic(&Testsuite);

    if (Testsuite.Informational.LastKnownPassedLocation.TestCaseName != 0)
        strcpy((char*)&lastTestCase, (char*)Testsuite.Informational.LastKnownPassedLocation.TestCaseName);
    if (Testsuite.Informational.LastKnownPassedLocation.TestSetName != 0)
        strcpy((char*)&lastTestSet, (char*)Testsuite.Informational.LastKnownPassedLocation.TestSetName);

}

void _EXIT exitTestSuite(void)
{
	utExit(&Testsuite);
}
```

### Program Logical/Infrastructure/AxisTemplate/AxisControl (IEC)

#### AxisControl.st - Init, cyclic, exit code
```iecst
//***********************************************************************
// Copyright: B&R Industrial Automation GmbH
// Author: B&R Industrial Automation GmbH
// Created: Jan 1, 2022
// Description: Tasks for axis control.
//***********************************************************************

PROGRAM _INIT

    ST_name(0, ADR(AxisControl.Status.TaskName), 0);

	// Inititialize mapp function blocks
	MpAlarmXCore_0.Enable := TRUE;
	MpAlarmXCore_0();
    ConfigurationInit;

    MpAxisBasic_0.Enable := TRUE;
	MpAxisBasic_0.MpLink := ADR(gAxisTemplate);
	MpAxisBasic_0();

    AxisInit;

END_PROGRAM

PROGRAM _CYCLIC

    MpAxisBasic_0.MpLink := ADR(gAxisTemplate);
    MC_BR_CheckRestorePositionData_0.Axis := ADR(gAxisTemplate);

	// Call all actions
    SimulationControl;
    AxisStateMachine;
    AxisCyclic;
	RecipeCyclic;

    // Assign MpLink
    MpAlarmXCore_0.MpLink := ADR(gAlarmXCore_AxisTemplate);

	// Call function block
	MpAlarmXCore_0();

END_PROGRAM

PROGRAM _EXIT

	// Disable the function blocls to unlink the MpLinks.
	// Do NOT disable MpAxisBasic, as this can cause problems during project transfer.
    MpRecipeRegPar_Par.Enable := FALSE;
	MpRecipeRegPar_Cfg.Enable := FALSE;
	MpAlarmXCore_0.Enable := FALSE;

	// Call function blocks
	MpRecipeRegPar_Par();
	MpRecipeRegPar_Cfg();
	MpAlarmXCore_0();

END_PROGRAM
```

#### AxisControl.typ - Local data types
```iecst
TYPE
	AxisSettingsType : 	STRUCT
		AxisFeatures : {REDUND_UNREPLICABLE} ARRAY[0..2]OF STRING[255];
		DriveConfiguration : {REDUND_UNREPLICABLE} McCfgPureVAxType;
		BaseConfiguration : {REDUND_UNREPLICABLE} McCfgAxType;
		BaseParam : {REDUND_UNREPLICABLE} McCfgAxMoveLimType;
	END_STRUCT;
	AxisMachineSettingsType : {REDUND_UNREPLICABLE} 	STRUCT
		ReferencePosition : {REDUND_UNREPLICABLE} LREAL := 0; (*[mm] Axis position after reference*)
	END_STRUCT;
	AxisControlCommandType : {REDUND_UNREPLICABLE} 	STRUCT
		UpdatePreviewParameters : {REDUND_UNREPLICABLE} BOOL;
		LoadRecipeParameters : {REDUND_UNREPLICABLE} BOOL;
		SaveRecipeParameters : {REDUND_UNREPLICABLE} BOOL;
		Power : {REDUND_UNREPLICABLE} BOOL;
		Reference : {REDUND_UNREPLICABLE} BOOL;
		MoveAbsolute : {REDUND_UNREPLICABLE} BOOL;
		MoveAdditive : {REDUND_UNREPLICABLE} BOOL;
		MoveToStart : {REDUND_UNREPLICABLE} BOOL;
		Abort : {REDUND_UNREPLICABLE} BOOL;
		Stop : {REDUND_UNREPLICABLE} BOOL;
		Reset : {REDUND_UNREPLICABLE} BOOL;
		JogPositive : {REDUND_UNREPLICABLE} BOOL;
		JogNegative : {REDUND_UNREPLICABLE} BOOL;
		Start : {REDUND_UNREPLICABLE} BOOL;
	END_STRUCT;
	AxisControlParametersType : {REDUND_UNREPLICABLE} 	STRUCT
		HomePosition : {REDUND_UNREPLICABLE} LREAL := 0; (*[mm] Home Position*)
		Position : {REDUND_UNREPLICABLE} LREAL := 0; (*[mm] Position for absolute move*)
		Distance : {REDUND_UNREPLICABLE} LREAL := 50; (*[mm] Distance for relative move*)
		Velocity : {REDUND_UNREPLICABLE} REAL := 100; (*[mm/s] Velocity for absoluate and relative moves*)
		Acceleration : {REDUND_UNREPLICABLE} REAL := 360; (*[mm/s2] Acceleration for absoluate and relative moves*)
		Deceleration : {REDUND_UNREPLICABLE} REAL := 360; (*[mm/s2] Deceleration for absoluate and relative moves*)
		JogVelocity : {REDUND_UNREPLICABLE} REAL := 100; (*[mm/s] Velocity used when jogging the axis*)
		StopDeceleration : {REDUND_UNREPLICABLE} REAL := 720; (*[mm/s2] Deceleration for stopping*)
	END_STRUCT;
	AxisControlStatusType : {REDUND_UNREPLICABLE} 	STRUCT
		TaskName : {REDUND_UNREPLICABLE} STRING[80];
		MachineSettingsName : {REDUND_UNREPLICABLE} STRING[255];
		ProductSettingsName : {REDUND_UNREPLICABLE} STRING[255];
		Status : {REDUND_UNREPLICABLE} STRING[80]; (*Machine Status*)
		IsReady : {REDUND_UNREPLICABLE} BOOL;
		ErrorActive : {REDUND_UNREPLICABLE} BOOL;
		Busy : {REDUND_UNREPLICABLE} BOOL;
		ReferenceRequired : {REDUND_UNREPLICABLE} BOOL;
		Position : {REDUND_UNREPLICABLE} LREAL;
		Velocity : {REDUND_UNREPLICABLE} REAL;
		Current : {REDUND_UNREPLICABLE} REAL;
		LagError : {REDUND_UNREPLICABLE} LREAL;
		MotorTemperature : {REDUND_UNREPLICABLE} REAL;
		IsHomed : {REDUND_UNREPLICABLE} BOOL;
		IsPowered : {REDUND_UNREPLICABLE} BOOL;
	END_STRUCT;
	AxisControlType : {REDUND_UNREPLICABLE} 	STRUCT
		Command : {REDUND_UNREPLICABLE} AxisControlCommandType;
		Parameters : {REDUND_UNREPLICABLE} AxisControlParametersType;
		Status : {REDUND_UNREPLICABLE} AxisControlStatusType;
	END_STRUCT;
	StateEnum :
		(
		STATE_INIT,
		STATE_POWER_ON,
		STATE_HOME,
		STATE_REFERENCE,
		STATE_MOVE_TO_HOME_POSITION,
		STATE_READY,
		STATE_MANUAL_OPERATION,
		STATE_AUTOMATIC_OPERATION,
		STATE_STOPPING,
		STATE_STOPPED,
		STATE_ABORTING,
		STATE_ABORTED,
		STATE_CLEARING,
		STATE_RESETTING
		);
	ParameterStateEnum :
		(
		PAR_STATE_INIT,
		PAR_STATE_READ,
		PAR_STATE_WRITE,
		PAR_STATE_READY
		);
	ConfigurationStateEnum :
		(
		CONFIG_STATE_INIT,
		CONFIG_STATE_READ,
		CONFIG_STATE_WRITE,
		CONFIG_STATE_READY
		);
	ManualStateEnum :
		(
		MANUAL_STATE_IDLE,
		MANUAL_STATE_JOG,
		MANUAL_STATE_MOVE,
		MANUAL_STATE_STOPPING
		);
	AutomaticStateEnum :
		(
		AUTOMATIC_STATE_IDLE,
		AUTOMATIC_STATE_RUNNING
		);
	AxisRecipeType : 	STRUCT
		EditDialogOpened : BOOL;
		CreateDialogOpened : BOOL;
		SaveRecipe : BOOL;
		LoadRecipe : BOOL;
		CreateRecipe : BOOL;
		State : AxisRecipeStepEnum;
		CategoryDropdown : STRING[50];
	END_STRUCT;
	AxisRecipeStepEnum :
		(
		REC_AXIS_WAIT,
		REC_AXIS_LOAD,
		REC_AXIS_SAVE,
		REC_AXIS_CREATE,
		REC_AXIS_STORE_MACH_SETTINGS,
		REC_AXIS_FACTORY_RESET
		);
END_TYPE
```

#### AxisControl.var - Local variables
```iecst
VAR
	i : {REDUND_UNREPLICABLE} USINT;
	RestorePosition : {REDUND_UNREPLICABLE} McAcpAxRestorePosType;
	ParameterState : {REDUND_UNREPLICABLE} ParameterStateEnum;
	ConfigurationState : {REDUND_UNREPLICABLE} ConfigurationStateEnum;
	State : {REDUND_UNREPLICABLE} StateEnum;
	AutomaticState : {REDUND_UNREPLICABLE} AutomaticStateEnum;
	ManualState : {REDUND_UNREPLICABLE} ManualStateEnum;
	AxisControl : {REDUND_UNREPLICABLE} AxisControlType;
	AxisSettings : {REDUND_UNREPLICABLE} AxisSettingsType;
END_VAR
(*Function Blocks*)
VAR
	MC_BR_CheckRestorePositionData_0 : {REDUND_UNREPLICABLE} MC_BR_CheckRestorePositionData;
	MpRecipeRegPar_Cfg : {REDUND_UNREPLICABLE} MpRecipeRegPar;
	MpRecipeRegPar_Par : {REDUND_UNREPLICABLE} MpRecipeRegPar;
	MpAlarmXCore_0 : {REDUND_UNREPLICABLE} MpAlarmXCore;
	MpAxisParameters : {REDUND_UNREPLICABLE} MpAxisBasicParType := (Distance:=70,Velocity:=100,Acceleration:=5000,Deceleration:=5000,Jog:=(Velocity:=70,Acceleration:=5000,Deceleration:=5000),AutoTune:=(MaxCurrentPercent:=50,MaxDistance:=720,MaxPositionError:=5));
	MpAxisBasic_0 : {REDUND_UNREPLICABLE} MpAxisBasic;
	MC_BR_ProcessConfig_AX : {REDUND_UNREPLICABLE} MC_BR_ProcessConfig; (*Function block to read and write the axis configuration*)
	MC_BR_ProcessConfig_ACP : {REDUND_UNREPLICABLE} MC_BR_ProcessConfig; (*Function block to read and write the ACOPOS configuration*)
	IsHomedEdgePos : {REDUND_UNREPLICABLE} R_TRIG;
	InPositionEdgePos : {REDUND_UNREPLICABLE} R_TRIG;
	ReferenceEdgePos : {REDUND_UNREPLICABLE} R_TRIG;
	MC_BR_ProcessParam_AX : {REDUND_UNREPLICABLE} MC_BR_ProcessParam; (*Function block to read and write the ACOPOS configuration*)
END_VAR
(*Recipe*)
VAR
	ParametersEdit : {REDUND_UNREPLICABLE} AxisControlParametersType;
	ParametersPreview : {REDUND_UNREPLICABLE} AxisControlParametersType;
	MachineSettings : {REDUND_UNREPLICABLE} AxisMachineSettingsType;
	MachineSettingsEdit : {REDUND_UNREPLICABLE} AxisMachineSettingsType;
	MachineSettingsPreview : {REDUND_UNREPLICABLE} AxisMachineSettingsType;
	AxisRecipe : {REDUND_UNREPLICABLE} AxisRecipeType;
END_VAR
```

#### Variables.var
```iecst
VAR
	MpAlarmXControlSpeedNotSetFB : MpAlarmXAlarmControl;
END_VAR
```

#### AxisStateMachine.st
```iecst
ACTION AxisStateMachine:

    InPositionEdgePos.CLK := MpAxisBasic_0.InPosition;
    InPositionEdgePos();
    IsHomedEdgePos.CLK := MpAxisBasic_0.IsHomed;
    IsHomedEdgePos();
    ReferenceEdgePos.CLK := AxisControl.Command.Reference;
    ReferenceEdgePos();

    CASE State OF
        STATE_STOPPING..STATE_RESETTING:
            // Nothing to do as we are already handling any stop or errors in these states

        ELSE
            IF ((MpAxisBasic_0.Error = TRUE) OR MpAlarmXCheckReaction(gMpLinkAlarmXCore, 'Error')) THEN
                // Check alarm reaction
                ResetAllAxisCommands;
                State := STATE_ABORTING;
            ELSIF ((AxisControl.Command.Power = FALSE) AND (State > STATE_POWER_ON)) THEN
                ResetAllAxisCommands;
                AxisControl.Status.Busy := TRUE;
                MpAxisBasic_0.Power := FALSE;
                State := STATE_POWER_ON;
            END_IF

    END_CASE

    CASE State OF

        STATE_INIT:
            AxisControl.Status.Status := 'Initializing';
            ChangeConfiguration;
			ChangeParameter;
            IF ((ConfigurationState = CONFIG_STATE_READY) AND (ParameterState = PAR_STATE_READY) AND (MpAxisBasic_0.Active = TRUE)) THEN
                AxisControl.Status.IsReady := TRUE;
                State := STATE_POWER_ON;
            END_IF

        STATE_POWER_ON:
            AxisControl.Status.Status := 'Waiting for power on';
            IF (MpAxisBasic_0.Info.ReadyToPowerOn = TRUE) THEN
                MpAxisBasic_0.Power := AxisControl.Command.Power;
            END_IF

            AxisControl.Status.Busy := MpAxisBasic_0.Power;
            IF (MpAxisBasic_0.PowerOn = TRUE) THEN
                MC_BR_CheckRestorePositionData_0.Execute := (MpAxisBasic_0.Info.HardwareInfo.Axis.AxisType <> mcAX_TYPE_PURE_VIRT);
                AxisControl.Status.Busy := FALSE;
                State := STATE_HOME;
            ELSE
                ChangeConfiguration;
            END_IF

        STATE_HOME:
            AxisControl.Status.Status := 'Waiting for home';
            IF ((MC_BR_CheckRestorePositionData_0.Done = TRUE) AND (MC_BR_CheckRestorePositionData_0.DataValid = TRUE)) THEN
                AxisControl.Status.ReferenceRequired := FALSE;
                MpAxisBasic_0.Home := TRUE;
                MpAxisParameters.Homing.Mode := mcHOMING_DEFAULT;
                AxisControl.Status.Busy := TRUE;
            ELSIF (MC_BR_CheckRestorePositionData_0.Busy = FALSE) THEN
                AxisControl.Status.ReferenceRequired := TRUE;
                State := STATE_REFERENCE;
            END_IF

            IF (MpAxisBasic_0.IsHomed = TRUE) THEN
                MC_BR_CheckRestorePositionData_0.Execute := FALSE;
                AxisControl.Status.ReferenceRequired := FALSE;
                AxisControl.Status.Busy := FALSE;
                AxisControl.Command.Reference := FALSE;
                MpAxisBasic_0.Home := FALSE;
                State := STATE_MOVE_TO_HOME_POSITION;
                ResetAllAxisCommands;
            END_IF

        STATE_REFERENCE:
            IF (AxisControl.Command.Reference = TRUE) THEN
                AxisControl.Command.Reference := FALSE;
                MpAxisBasic_0.Home := TRUE;
                AxisControl.Status.Busy := TRUE;
                MpAxisParameters.Homing.Mode := mcHOMING_DIRECT;
                MpAxisParameters.Homing.Position := MachineSettings.ReferencePosition;
            END_IF

            IF (IsHomedEdgePos.Q  = TRUE) THEN
                MC_BR_CheckRestorePositionData_0.Execute := FALSE;
                AxisControl.Status.ReferenceRequired := FALSE;
                MpAxisBasic_0.Home := FALSE;
                State := STATE_MOVE_TO_HOME_POSITION;
                ResetAllAxisCommands;
            END_IF

        STATE_MOVE_TO_HOME_POSITION:
            AxisControl.Status.Status := 'Moving to home position';
            MpAxisParameters.Position := AxisControl.Parameters.HomePosition;
            MpAxisParameters.Direction := mcDIR_SHORTEST_WAY;
            MpAxisBasic_0.MoveAbsolute := TRUE;
            IF (InPositionEdgePos.Q  = TRUE) THEN
                AxisControl.Status.Busy := FALSE;
                MpAxisBasic_0.MoveAbsolute := FALSE;
                State := STATE_READY;
            END_IF

        // In this State the module is error free and ready for a command (manual or automatic)
        STATE_READY:
            AxisControl.Status.Status := 'Ready';
            AxisControl.Status.Busy := FALSE;
            IF (ReferenceEdgePos.Q = TRUE) THEN
                State := STATE_REFERENCE;
            ELSIF ((MpAlarmXCheckReaction(gMpLinkAlarmXCore, 'Warning') = FALSE) AND (AutomaticCommand(AxisControl.Command) = TRUE)) THEN
                State := STATE_AUTOMATIC_OPERATION;
            ELSIF (ManualCommand(AxisControl.Command) = TRUE) THEN
                State := STATE_MANUAL_OPERATION;
            END_IF

        STATE_MANUAL_OPERATION:
            AxisControl.Status.Status := 'Manual running';
            AxisControl.Status.Busy := TRUE;
            AxisManual;

        STATE_AUTOMATIC_OPERATION:
            AxisControl.Status.Status := 'Automatic running';
            AxisControl.Status.Busy := TRUE;
            IF MpAlarmXCheckReaction(gMpLinkAlarmXCore, 'Error') THEN
                AxisControl.Command.Stop := TRUE;
            END_IF

            AxisAutomatic;

        // In this State the module will attempt to bring the axis to a controlled stop.
        STATE_STOPPING:
            AxisControl.Status.Status := 'Stopping';

            // Stop the axis if it is powered on
            MpAxisBasic_0.Stop := MpAxisBasic_0.PowerOn;
            MpAxisParameters.Deceleration := AxisControl.Parameters.StopDeceleration;
            IF ((MpAxisBasic_0.PowerOn = FALSE) OR (MpAxisBasic_0.Stopped = TRUE)) THEN
                MpAxisBasic_0.Stop := FALSE;
                State := STATE_STOPPED;
            END_IF

        // In this State the module is powered on and at standstill.
        STATE_STOPPED:
            State := STATE_RESETTING;

        // In this State the module will bring the axis to a rapid stop
        STATE_ABORTING:
            MpAxisParameters.Stop.Deceleration := 0;
            MpAxisBasic_0.Stop := MpAxisBasic_0.PowerOn;
            IF ((MpAxisBasic_0.PowerOn = FALSE) OR (MpAxisBasic_0.Stopped = TRUE)) THEN
                MpAxisBasic_0.Stop := FALSE;
                IF (MpAlarmXCheckReaction(gMpLinkAlarmXCore, 'SafetyError') = TRUE) THEN
                    // Safety errors also power off the axis
                    MpAxisBasic_0.Power := FALSE;
                    IF (MpAxisBasic_0.PowerOn = FALSE) THEN
                        State := STATE_ABORTED;
                    END_IF
                ELSE
                    State := STATE_ABORTED;
                END_IF
            END_IF

        STATE_ABORTED:
            State := STATE_CLEARING;

        STATE_CLEARING:
            State := STATE_RESETTING;

        // In this State the module attempts to clear any outstanding errors.  No hazardous motion should occur in this State.
        STATE_RESETTING:
            ResetAllAxisCommands;
            IF (AxisControl.Command.Reset = TRUE) THEN
                AxisControl.Status.Busy := TRUE;
                AxisControl.Command.Reset := FALSE;
                MpAxisBasic_0.ErrorReset := TRUE;
                AxisReset;
            ELSE
                MpAxisBasic_0.ErrorReset := FALSE;
            END_IF

            IF ((MpAxisBasic_0.Error = FALSE) AND (MpAlarmXCheckReaction(gMpLinkAlarmXCore, 'Error') = FALSE)) THEN
                AxisControl.Status.Busy := FALSE;
                IF (MpAxisBasic_0.PowerOn = FALSE) THEN
                    State := STATE_POWER_ON;
                ELSIF (MpAxisBasic_0.IsHomed = TRUE) THEN
                    State := STATE_READY;
                ELSE
                    State := STATE_HOME;
                END_IF
            END_IF

    END_CASE

    MpAxisBasic_0.Parameters := ADR(MpAxisParameters);
    MpAxisBasic_0();

    MC_BR_CheckRestorePositionData_0.DataAddress := ADR(RestorePosition);
    MC_BR_CheckRestorePositionData_0();

    AxisControl.Status.ErrorActive := MpAxisBasic_0.Error;
    AxisControl.Status.IsHomed := MpAxisBasic_0.IsHomed;
    AxisControl.Status.IsPowered := MpAxisBasic_0.PowerOn;
    AxisControl.Status.Position := MpAxisBasic_0.Position;
    AxisControl.Status.Velocity := MpAxisBasic_0.Velocity;

END_ACTION

ACTION ResetAllAxisCommands:

    MpAxisBasic_0.MoveAbsolute := FALSE;
    MpAxisBasic_0.MoveAdditive := FALSE;
    MpAxisBasic_0.MoveVelocity := FALSE;
    MpAxisBasic_0.ReleaseBrake := FALSE;
    MpAxisBasic_0.ErrorReset := FALSE;
    MpAxisBasic_0.JogPositive := FALSE;
    MpAxisBasic_0.JogNegative := FALSE;

END_ACTION
```

#### AxisControlModes.st
```iecst
ACTION AxisInit:

END_ACTION

ACTION AxisCyclic:

    IF (MpRecipeRegPar_Par.UpdateNotification) THEN

    END_IF

END_ACTION

ACTION AxisManual:

    MpAxisParameters.Jog.Velocity := AxisControl.Parameters.JogVelocity;
    MpAxisParameters.Position := AxisControl.Parameters.Position;
    MpAxisParameters.Distance := AxisControl.Parameters.Distance;
    MpAxisParameters.Acceleration := AxisControl.Parameters.Acceleration;
    MpAxisParameters.Deceleration := AxisControl.Parameters.Deceleration;

    CASE ManualState OF
        MANUAL_STATE_IDLE:
            IF ((AxisControl.Command.JogNegative = TRUE) OR (AxisControl.Command.JogPositive = TRUE)) THEN
                ManualState := MANUAL_STATE_JOG;
            ELSIF ((AxisControl.Command.MoveAbsolute = TRUE) OR (AxisControl.Command.MoveAdditive = TRUE)) THEN
                MpAxisBasic_0.MoveAbsolute := AxisControl.Command.MoveAbsolute;
                MpAxisBasic_0.MoveAdditive := AxisControl.Command.MoveAdditive;
                AxisControl.Command.MoveAbsolute := FALSE;
                AxisControl.Command.MoveAdditive := FALSE;
                ManualState := MANUAL_STATE_MOVE;
            END_IF

        MANUAL_STATE_JOG:
            MpAxisBasic_0.JogNegative := AxisControl.Command.JogNegative;
            MpAxisBasic_0.JogPositive := AxisControl.Command.JogPositive;
            IF (AxisControl.Command.Stop = TRUE) THEN
                AxisControl.Command.Stop := FALSE;
                MpAxisBasic_0.Stop := TRUE;
                ManualState := MANUAL_STATE_STOPPING;
            ELSIF ((AxisControl.Command.JogNegative = FALSE) AND (AxisControl.Command.JogPositive = FALSE)) THEN
                MpAxisBasic_0.Stop := FALSE;
                MpAxisBasic_0.JogPositive := FALSE;
                MpAxisBasic_0.JogNegative := FALSE;
                ManualState := MANUAL_STATE_STOPPING;
            END_IF

        MANUAL_STATE_MOVE:
            IF (AxisControl.Command.Stop = TRUE) THEN
                MpAxisBasic_0.MoveAbsolute := FALSE;
                MpAxisBasic_0.MoveAdditive := FALSE;
                AxisControl.Command.Stop := FALSE;
                MpAxisBasic_0.Stop := TRUE;
                ManualState := MANUAL_STATE_STOPPING;
            ELSIF (InPositionEdgePos.Q = TRUE) THEN
                MpAxisBasic_0.MoveAbsolute := FALSE;
                MpAxisBasic_0.MoveAdditive := FALSE;
                ManualState := MANUAL_STATE_IDLE;
                state := STATE_READY;
            ELSIF ((AxisControl.Command.JogNegative = TRUE) OR (AxisControl.Command.JogPositive = TRUE)) THEN
                MpAxisBasic_0.MoveAbsolute := FALSE;
                MpAxisBasic_0.MoveAdditive := FALSE;
                ManualState := MANUAL_STATE_JOG;
            END_IF

        MANUAL_STATE_STOPPING:
            MpAxisBasic_0.JogNegative := FALSE;
            MpAxisBasic_0.JogPositive := FALSE;
            MpAxisBasic_0.MoveAbsolute := FALSE;
            MpAxisBasic_0.MoveAdditive := FALSE;

            IF (MpAxisBasic_0.MoveActive = FALSE) THEN
                ManualState := MANUAL_STATE_IDLE;
                state := STATE_READY;
            END_IF
    END_CASE

END_ACTION

ACTION AxisAutomatic:

    CASE AutomaticState OF
        AUTOMATIC_STATE_IDLE:
            IF (AxisControl.Command.Start = TRUE) THEN
                MpAlarmXControlSpeedNotSetFB.Set := (MpAxisParameters.Velocity = 0);
                AxisControl.Command.Start := FALSE;
                AutomaticState := AUTOMATIC_STATE_RUNNING;
            END_IF

        AUTOMATIC_STATE_RUNNING:
            MpAxisBasic_0.MoveVelocity := TRUE;
            MpAxisParameters.Velocity := AxisControl.Parameters.Velocity;
            MpAxisParameters.Acceleration := AxisControl.Parameters.Acceleration;
            MpAxisParameters.Deceleration := AxisControl.Parameters.Deceleration;

            IF (AxisControl.Command.Stop = TRUE) THEN
                AxisControl.Command.Stop := FALSE;
                MpAxisBasic_0.MoveVelocity := FALSE;
                state := STATE_READY;
                AutomaticState := AUTOMATIC_STATE_IDLE;
            END_IF
    END_CASE

END_ACTION

ACTION AxisReset:

END_ACTION
```

#### Recipe.st
```iecst
ACTION RecipeInit:

    // Register the variables with the recipe system
    AxisControl.Status.ProductSettingsName := AxisControl.Status.TaskName;
    brsstrcat(ADR(AxisControl.Status.ProductSettingsName), ADR(':ParametersPreview'));
    MpRecipeRegPar_Par.MpLink := ADR(gMpLinkRecipeXml);
    MpRecipeRegPar_Par.Enable := TRUE;
    MpRecipeRegPar_Par.PVName := ADR(AxisControl.Status.ProductSettingsName);
    MpRecipeRegPar_Par.Category := ADR(PRODUCT_CATEGORY);
    MpRecipeRegPar_Par();
    ParametersPreview;
    ParametersEdit;

    AxisControl.Status.MachineSettingsName := AxisControl.Status.TaskName;
    brsstrcat(ADR(AxisControl.Status.MachineSettingsName), ADR(':MachineSettingsPreview'));
    MpRecipeRegPar_Cfg.MpLink := ADR(gMpLinkRecipeXml);
    MpRecipeRegPar_Cfg.Enable := TRUE;
    MpRecipeRegPar_Cfg.PVName := ADR(AxisControl.Status.MachineSettingsName);
    MpRecipeRegPar_Cfg.Category := ADR(MACHINE_CATEGORY);
    MpRecipeRegPar_Cfg();
    MachineSettingsPreview;
    MachineSettingsEdit;

    // Activate RegPar FUBs
    WHILE NOT(MpRecipeRegPar_Par.Active OR MpRecipeRegPar_Par.Error) DO
        MpRecipeRegPar_Par();
    END_WHILE
    WHILE NOT(MpRecipeRegPar_Cfg.Active OR MpRecipeRegPar_Cfg.Error) DO
        MpRecipeRegPar_Cfg();
    END_WHILE

END_ACTION

ACTION RecipeCyclic:

	IF (AxisRecipe.EditDialogOpened OR AxisRecipe.CreateDialogOpened) THEN
		IF (brsstrcmp(ADR(AxisRecipe.CategoryDropdown), ADR('Product')) = 0) THEN
			ParametersEdit := ParametersPreview;
		ELSIF (brsstrcmp(ADR(AxisRecipe.CategoryDropdown), ADR('Machine')) = 0) THEN
			MachineSettingsEdit := MachineSettingsPreview;
		END_IF
		AxisRecipe.EditDialogOpened := FALSE;
		AxisRecipe.CreateDialogOpened := FALSE;
	END_IF

	CASE AxisRecipe.State OF
		REC_AXIS_WAIT:
			IF AxisRecipe.CreateRecipe THEN
				AxisRecipe.State := REC_AXIS_CREATE;
				AxisRecipe.CreateRecipe := FALSE;
			ELSIF AxisRecipe.SaveRecipe THEN
				AxisRecipe.State := REC_AXIS_SAVE;
				AxisRecipe.SaveRecipe := FALSE;
			ELSIF AxisRecipe.LoadRecipe THEN
				AxisRecipe.State := REC_AXIS_LOAD;
				AxisRecipe.LoadRecipe := FALSE;
			END_IF

		REC_AXIS_CREATE:
			IF (brsstrcmp(ADR(AxisRecipe.CategoryDropdown), ADR('Product')) = 0) THEN
				ParametersPreview := ParametersEdit;
			ELSIF (brsstrcmp(ADR(AxisRecipe.CategoryDropdown), ADR('Machine')) = 0) THEN
				MachineSettingsPreview := MachineSettingsEdit;
			END_IF
			AxisRecipe.State := REC_AXIS_WAIT;

		REC_AXIS_LOAD:
			IF (brsstrcmp(ADR(AxisRecipe.CategoryDropdown), ADR('Product')) = 0) THEN
				AxisControl.Parameters := ParametersPreview;
			ELSIF (brsstrcmp(ADR(AxisRecipe.CategoryDropdown), ADR('Machine')) = 0) THEN
				MachineSettings := MachineSettingsPreview;
			END_IF
			AxisRecipe.State := REC_AXIS_WAIT;

		REC_AXIS_SAVE:
			IF (brsstrcmp(ADR(AxisRecipe.CategoryDropdown), ADR('Product')) = 0) THEN
				ParametersPreview := ParametersEdit;
			ELSIF (brsstrcmp(ADR(AxisRecipe.CategoryDropdown), ADR('Machine')) = 0) THEN
				MachineSettingsPreview := MachineSettingsEdit;
			END_IF
			AxisRecipe.State := REC_AXIS_WAIT;

	END_CASE;

	MpRecipeRegPar_Par.MpLink := ADR(gMpLinkRecipeXml);
	MpRecipeRegPar_Par();

	MpRecipeRegPar_Cfg.MpLink := ADR(gMpLinkRecipeXml);
	MpRecipeRegPar_Cfg();

END_ACTION
```

#### SimulationControl.st
```iecst
ACTION SimulationControl:

    IF NOT (DiagCpuIsARsim() OR DiagCpuIsSimulated()) THEN
        RETURN;
    END_IF

    IF ((MpAxisBasic_0.IsHomed = FALSE) AND (MpAxisBasic_0.Home = FALSE)) THEN
        AxisControl.Command.Reference := TRUE;
    END_IF

END_ACTION
```

#### ManualCommand.st
```iecst
// Returns True if a manual command is active, false otherwise
FUNCTION ManualCommand
    ManualCommand := Commands.JogNegative OR Commands.JogPositive OR Commands.MoveAbsolute OR Commands.MoveAdditive;
END_FUNCTION
```

#### AutomaticCommand.st
```iecst
// Returns True if an automatic command is active
FUNCTION AutomaticCommand

    AutomaticCommand := Commands.Start;

END_FUNCTION
```

#### ChangeConfiguration.st
```iecst
ACTION ConfigurationInit:

    AxisSettings.DriveConfiguration.PureVirtualAxis.AxisFeatures.FeatureReference.DataAddress := ADR(AxisSettings.AxisFeatures);
    AxisSettings.DriveConfiguration.PureVirtualAxis.AxisFeatures.FeatureReference.NumberOfArrayElements := SIZEOF(AxisSettings.AxisFeatures)/SIZEOF(AxisSettings.AxisFeatures[0]);
    AxisSettings.DriveConfiguration.PureVirtualAxis.AxisFeatures.FeatureReference.NumberOfElements := 0;
    i := 0;
    WHILE ((i <= SIZEOF(AxisSettings.AxisFeatures)/SIZEOF(AxisSettings.AxisFeatures[0])) AND (AxisSettings.AxisFeatures[i] <> '')) DO
        i := i + 1;
    END_WHILE
    AxisSettings.DriveConfiguration.PureVirtualAxis.AxisFeatures.FeatureReference.NumberOfElements := i;

    MC_BR_ProcessConfig_AX.DataAddress := ADR(AxisSettings.BaseConfiguration);
    MC_BR_ProcessConfig_AX.DataType := mcCFG_AX;

    MC_BR_ProcessConfig_ACP.DataAddress := ADR(AxisSettings.DriveConfiguration);
    MC_BR_ProcessConfig_ACP.DataType := mcCFG_PURE_V_AX;

    ConfigurationState := CONFIG_STATE_INIT;

END_ACTION

ACTION ChangeConfiguration:

    CASE ConfigurationState OF
        CONFIG_STATE_INIT:

            // Build up the string for the name
            MC_BR_ProcessConfig_ACP.Name := MpAxisBasic_0.Info.HardwareInfo.Axis.ConfigElementLocation;
            MC_BR_ProcessConfig_AX.Name := MpAxisBasic_0.Info.HardwareInfo.Axis.AxisName;

            IF (MpAxisBasic_0.Active = TRUE) THEN
                ConfigurationState := CONFIG_STATE_READ;
            END_IF

        CONFIG_STATE_READ:
            MC_BR_ProcessConfig_ACP.Mode := mcPCM_LOAD;
            MC_BR_ProcessConfig_ACP.Execute := TRUE;

            MC_BR_ProcessConfig_AX.Mode := mcPCM_LOAD;
            MC_BR_ProcessConfig_AX.Execute := TRUE;
            IF (MC_BR_ProcessConfig_ACP.Done = TRUE) AND (MC_BR_ProcessConfig_AX.Done = TRUE) THEN
                MC_BR_ProcessConfig_ACP.Execute := FALSE;
                MC_BR_ProcessConfig_AX.Execute := FALSE;
                ConfigurationState := CONFIG_STATE_READY;
            END_IF

        CONFIG_STATE_WRITE:
            MC_BR_ProcessConfig_ACP.Mode := mcPCM_SAVE;
            MC_BR_ProcessConfig_ACP.Execute := TRUE;

            MC_BR_ProcessConfig_AX.Mode := mcPCM_SAVE;
            MC_BR_ProcessConfig_AX.Execute := TRUE;
            IF (MC_BR_ProcessConfig_ACP.Done = TRUE) AND (MC_BR_ProcessConfig_AX.Done = TRUE) THEN
                MC_BR_ProcessConfig_ACP.Execute := FALSE;
                MC_BR_ProcessConfig_AX.Execute := FALSE;
                ConfigurationState := CONFIG_STATE_READY;
            END_IF

        CONFIG_STATE_READY:

    END_CASE

    MC_BR_ProcessConfig_ACP();
    MC_BR_ProcessConfig_AX();

END_ACTION

ACTION ParameterInit:

	MC_BR_ProcessParam_AX.DataAddress := ADR(AxisSettings.BaseParam);
    MC_BR_ProcessParam_AX.DataType := mcCFG_AX_MOVE_LIM;

    ParameterState := PAR_STATE_INIT;

END_ACTION

ACTION ChangeParameter:

    CASE ParameterState OF
        PAR_STATE_INIT:

            MC_BR_ProcessParam_AX.Component := MpAxisBasic_0.MpLink;

            IF (MpAxisBasic_0.Active = TRUE) THEN
                ParameterState := PAR_STATE_READ;
            END_IF

        PAR_STATE_READ:
            MC_BR_ProcessParam_AX.Mode := mcPPM_READ;
            MC_BR_ProcessParam_AX.Execute := TRUE;

            IF (MC_BR_ProcessParam_AX.Done = TRUE) THEN
                MC_BR_ProcessParam_AX.Execute := FALSE;
                ParameterState := PAR_STATE_READY;
            END_IF

        PAR_STATE_WRITE:
            MC_BR_ProcessParam_AX.Mode := mcPPM_WRITE;
            MC_BR_ProcessParam_AX.Execute := TRUE;

            IF (MC_BR_ProcessParam_AX.Done = TRUE) THEN
                MC_BR_ProcessParam_AX.Execute := FALSE;
                ParameterState := PAR_STATE_READY;
            END_IF

        PAR_STATE_READY:

    END_CASE

    MC_BR_ProcessParam_AX();

END_ACTION
```

#### Types.typ - not listed in the package file held
```iecst
TYPE
	AxisMachineSettingsType : {REDUND_UNREPLICABLE} 	STRUCT
		ReferencePosition : {REDUND_UNREPLICABLE} LREAL := 0.0; (*[mm] Position when the axis is referenced*)
		AxisFeatures : {REDUND_UNREPLICABLE} ARRAY[0..4]OF STRING[255] := ['CamAut_cutting','ValueSource','',2('')];
		DriveConfiguration : {REDUND_UNREPLICABLE} McCfgPureVAxType;
		BaseConfiguration : {REDUND_UNREPLICABLE} McCfgAxType;
	END_STRUCT;
	AxisControlCommandType : {REDUND_UNREPLICABLE} 	STRUCT
		UpdatePreviewParameters : {REDUND_UNREPLICABLE} BOOL;
		ResetEditParameters : {REDUND_UNREPLICABLE} BOOL;
		Power : {REDUND_UNREPLICABLE} BOOL;
		Reference : {REDUND_UNREPLICABLE} BOOL;
		MoveAbsolute : {REDUND_UNREPLICABLE} BOOL;
		MoveAdditive : {REDUND_UNREPLICABLE} BOOL;
		MoveToStart : {REDUND_UNREPLICABLE} BOOL;
		Abort : {REDUND_UNREPLICABLE} BOOL;
		Stop : {REDUND_UNREPLICABLE} BOOL;
		Reset : {REDUND_UNREPLICABLE} BOOL;
		JogPositive : {REDUND_UNREPLICABLE} BOOL;
		JogNegative : {REDUND_UNREPLICABLE} BOOL;
		Start : {REDUND_UNREPLICABLE} BOOL;
	END_STRUCT;
	AxisControlParametersType : {REDUND_UNREPLICABLE} 	STRUCT
		HomePosition : {REDUND_UNREPLICABLE} LREAL := 0; (*[mm] Home Position*)
		Position : {REDUND_UNREPLICABLE} LREAL := 0; (*[mm] Position for absolute move*)
		Distance : {REDUND_UNREPLICABLE} LREAL := 50; (*[mm] Distance for relative move*)
		Velocity : {REDUND_UNREPLICABLE} REAL := 100; (*[mm/s] Velocity for absoluate and relative moves*)
		Acceleration : {REDUND_UNREPLICABLE} REAL := 360; (*[mm/s2] Acceleration for absoluate and relative moves*)
		Deceleration : {REDUND_UNREPLICABLE} REAL := 360; (*[mm/s2] Deceleration for absoluate and relative moves*)
		JogVelocity : {REDUND_UNREPLICABLE} REAL := 100; (*[mm/s] Velocity used when jogging the axis*)
		StopDeceleration : {REDUND_UNREPLICABLE} REAL := 720; (*[mm/s2] Deceleration for stopping*)
	END_STRUCT;
	AxisControlStatusType : {REDUND_UNREPLICABLE} 	STRUCT
		TaskName : {REDUND_UNREPLICABLE} STRING[80];
		MachineSettingsName : {REDUND_UNREPLICABLE} STRING[255];
		ProductSettingsName : {REDUND_UNREPLICABLE} STRING[255];
		ProductPreviewSettingsName : {REDUND_UNREPLICABLE} STRING[255];
		Status : {REDUND_UNREPLICABLE} STRING[80]; (*Machine Status*)
		IsReady : {REDUND_UNREPLICABLE} BOOL;
		ErrorActive : {REDUND_UNREPLICABLE} BOOL;
		Busy : {REDUND_UNREPLICABLE} BOOL;
		ReferenceRequired : {REDUND_UNREPLICABLE} BOOL;
		Position : {REDUND_UNREPLICABLE} LREAL;
		Velocity : {REDUND_UNREPLICABLE} REAL;
		Current : {REDUND_UNREPLICABLE} REAL;
		LagError : {REDUND_UNREPLICABLE} LREAL;
		MotorTemperature : {REDUND_UNREPLICABLE} REAL;
		IsHomed : {REDUND_UNREPLICABLE} BOOL;
		IsPowered : {REDUND_UNREPLICABLE} BOOL;
	END_STRUCT;
	AxisControlType : {REDUND_UNREPLICABLE} 	STRUCT
		Command : {REDUND_UNREPLICABLE} AxisControlCommandType;
		Parameters : {REDUND_UNREPLICABLE} AxisControlParametersType;
		Status : {REDUND_UNREPLICABLE} AxisControlStatusType;
	END_STRUCT;
	stateEnum :
		(
		STATE_INIT,
		STATE_POWER_ON,
		STATE_HOME,
		STATE_REFERENCE,
		STATE_MOVE_TO_HOME_POSITION,
		STATE_READY,
		STATE_MANUAL_OPERATION,
		STATE_AUTOMATIC_OPERATION,
		STATE_STOPPING,
		STATE_STOPPED,
		STATE_ABORTING,
		STATE_ABORTED,
		STATE_CLEARING,
		STATE_RESETTING
		);
	configurationStateEnum :
		(
		CONFIG_STATE_INIT,
		CONFIG_STATE_READ,
		CONFIG_STATE_WRITE,
		CONFIG_STATE_READY
		);
	manualStateEnum :
		(
		MANUAL_STATE_IDLE,
		MANUAL_STATE_JOG,
		MANUAL_STATE_MOVE,
		MANUAL_STATE_STOPPING
		);
END_TYPE
```

#### AxisStandard.var - not listed in the package file held
```iecst
VAR
	i : {REDUND_UNREPLICABLE} USINT;
	restorePosition : {REDUND_UNREPLICABLE} McAcpAxRestorePosType;
	MC_BR_CheckRestorePositionDataFB : {REDUND_UNREPLICABLE} MC_BR_CheckRestorePositionData;
	MpRecipeRegPar_MachineFB : {REDUND_UNREPLICABLE} MpRecipeRegPar;
	MpRecipeRegPar_UserFB : {REDUND_UNREPLICABLE} MpRecipeRegPar;
	MpRecipeRegPar_PreFB : {REDUND_UNREPLICABLE} MpRecipeRegPar; (*Register preview parameters*)
	MpRecipeRegPar_UserPreFB : {REDUND_UNREPLICABLE} MpRecipeRegPar; (*Register preview parameters*)
	MpAlarmXCoreFB : {REDUND_UNREPLICABLE} MpAlarmXCore;
	MpAxisParameters : {REDUND_UNREPLICABLE} MpAxisBasicParType := (Distance:=70,Velocity:=100,Acceleration:=5000,Deceleration:=5000,Jog:=(Velocity:=70,Acceleration:=5000,Deceleration:=5000),AutoTune:=(MaxCurrentPercent:=50,MaxDistance:=720,MaxPositionError:=5));
	MpAxisBasicFB : {REDUND_UNREPLICABLE} MpAxisBasic;
	MC_BR_ProcessConfig_AX : {REDUND_UNREPLICABLE} MC_BR_ProcessConfig; (*Function block to read and write the axis configuration*)
	MC_BR_ProcessConfig_ACP : {REDUND_UNREPLICABLE} MC_BR_ProcessConfig; (*Function block to read and write the ACOPOS configuration*)
	configurationState : {REDUND_UNREPLICABLE} configurationStateEnum;
	state : {REDUND_UNREPLICABLE} stateEnum;
	AutomaticState : {REDUND_UNREPLICABLE} USINT;
	ManualState : {REDUND_UNREPLICABLE} USINT;
	MachineSettings : {REDUND_UNREPLICABLE} AxisMachineSettingsType;
	PreviewParameters : {REDUND_UNREPLICABLE} AxisControlParametersType;
	AxisControl : {REDUND_UNREPLICABLE} AxisControlType;
	IsHomedEdgePos : {REDUND_UNREPLICABLE} R_TRIG;
	InPositionEdgePos : {REDUND_UNREPLICABLE} R_TRIG;
	ReferenceEdgePos : {REDUND_UNREPLICABLE} R_TRIG;
END_VAR
```
